C09046=1041.866,-97.475,-73.988,168.955,34.986,156.606
C09047=1041.872,-97.226,-73.998,168.958,34.986,156.606
C09048=1041.878,-96.977,-74.009,168.960,34.986,156.606
C09049=1041.883,-96.727,-74.019,168.962,34.986,156.606
C09050=1041.890,-96.477,-74.030,168.965,34.986,156.606
C09051=1041.895,-96.227,-74.040,168.967,34.986,156.606
C09052=1041.902,-95.978,-74.050,168.970,34.987,156.606
C09053=1041.908,-95.728,-74.061,168.972,34.987,156.606
C09054=1041.914,-95.478,-74.071,168.974,34.987,156.606
C09055=1041.920,-95.229,-74.082,168.977,34.987,156.606
C09056=1041.926,-94.979,-74.093,168.979,34.987,156.606
C09057=1041.932,-94.729,-74.102,168.982,34.987,156.606
C09058=1041.938,-94.479,-74.113,168.984,34.987,156.606
C09059=1041.945,-94.230,-74.124,168.986,34.987,156.606
C09060=1041.950,-93.980,-74.134,168.989,34.987,156.606
C09061=1041.956,-93.730,-74.145,168.991,34.987,156.606
C09062=1041.962,-93.481,-74.155,168.994,34.988,156.606
C09063=1041.969,-93.230,-74.165,168.996,34.988,156.606
C09064=1041.975,-92.981,-74.176,168.998,34.988,156.606
C09065=1041.981,-92.732,-74.187,169.001,34.988,156.606
C09066=1041.986,-92.482,-74.197,169.003,34.988,156.606
C09067=1041.993,-92.232,-74.207,169.006,34.988,156.606
C09068=1041.999,-91.982,-74.218,169.008,34.988,156.606
C09069=1042.005,-91.733,-74.229,169.011,34.988,156.606
C09070=1042.011,-91.484,-74.239,169.013,34.988,156.606
C09071=1042.017,-91.233,-74.250,169.015,34.988,156.606
C09072=1042.024,-90.984,-74.260,169.018,34.989,156.606
C09073=1042.029,-90.734,-74.271,169.020,34.989,156.606
C09074=1042.036,-90.485,-74.281,169.023,34.989,156.606
C09075=1042.042,-90.235,-74.293,169.025,34.989,156.606
C09076=1042.048,-89.985,-74.303,169.027,34.990,156.606
C09077=1042.054,-89.735,-74.313,169.030,34.990,156.606
C09078=1042.061,-89.485,-74.324,169.032,34.990,156.606
C09079=1042.066,-89.236,-74.335,169.034,34.990,156.606
C09080=1042.073,-88.987,-74.346,169.037,34.990,156.606
C09081=1042.079,-88.736,-74.357,169.039,34.990,156.606
C09082=1042.085,-88.487,-74.366,169.042,34.990,156.606
C09083=1042.091,-88.237,-74.377,169.044,34.990,156.606
C09084=1042.097,-87.987,-74.388,169.046,34.990,156.606
C09085=1042.104,-87.738,-74.399,169.049,34.991,156.606
C09086=1042.110,-87.488,-74.410,169.051,34.991,156.606
C09087=1042.116,-87.238,-74.421,169.054,34.991,156.606
C09088=1042.122,-86.989,-74.431,169.056,34.991,156.606
C09089=1042.128,-86.739,-74.442,169.058,34.991,156.606
C09090=1042.134,-86.489,-74.453,169.061,34.992,156.606
C09091=1042.141,-86.240,-74.464,169.063,34.992,156.606
C09092=1042.147,-85.991,-74.474,169.066,34.992,156.606
C09093=1042.153,-85.740,-74.486,169.068,34.992,156.606
C09094=1042.159,-85.491,-74.496,169.070,34.993,156.606
C09095=1042.166,-85.240,-74.506,169.073,34.993,156.606
C09096=1042.171,-84.991,-74.517,169.075,34.993,156.606
C09097=1042.178,-84.742,-74.528,169.077,34.993,156.606
C09098=1042.184,-84.492,-74.539,169.079,34.993,156.605
C09099=1042.190,-84.242,-74.550,169.081,34.993,156.605
C09100=1042.197,-83.957,-74.563,169.085,34.994,156.606
C09101=1042.204,-83.673,-74.575,169.087,34.994,156.606
C09102=1042.211,-83.387,-74.587,169.089,34.994,156.606
C09103=1042.219,-83.103,-74.600,169.092,34.994,156.605
C09104=1042.225,-82.853,-74.611,169.094,34.994,156.605
C09105=1042.231,-82.604,-74.621,169.097,34.995,156.606
C09106=1042.238,-82.354,-74.632,169.099,34.995,156.606
C09107=1042.243,-82.104,-74.643,169.102,34.995,156.605
C09108=1042.250,-81.854,-74.654,169.104,34.995,156.605
C09109=1042.256,-81.605,-74.665,169.106,34.995,156.605
C09110=1042.263,-81.355,-74.676,169.109,34.995,156.605
C09111=1042.269,-81.106,-74.686,169.111,34.996,156.606
C09112=1042.276,-80.856,-74.698,169.113,34.996,156.606
C09113=1042.281,-80.606,-74.709,169.116,34.996,156.605
C09114=1042.288,-80.356,-74.720,169.118,34.996,156.605
C09115=1042.294,-80.107,-74.731,169.121,34.997,156.606
C09116=1042.301,-79.857,-74.742,169.123,34.997,156.606
C09117=1042.306,-79.607,-74.753,169.125,34.997,156.606
C09118=1042.313,-79.357,-74.764,169.128,34.997,156.605
C09119=1042.319,-79.108,-74.776,169.130,34.998,156.606
C09120=1042.325,-78.858,-74.787,169.132,34.998,156.606
C09121=1042.331,-78.609,-74.798,169.135,34.999,156.606
C09122=1042.337,-78.358,-74.809,169.137,34.999,156.606
C09123=1042.343,-78.110,-74.821,169.139,34.999,156.606
C09124=1042.350,-77.859,-74.832,169.142,35.000,156.606
C09125=1042.356,-77.610,-74.842,169.144,35.000,156.606
C09126=1042.362,-77.360,-74.853,169.146,35.000,156.606
C09127=1042.368,-77.111,-74.865,169.149,35.001,156.606
C09128=1042.375,-76.861,-74.876,169.151,35.001,156.606
C09129=1042.381,-76.611,-74.887,169.153,35.002,156.606
C09130=1042.387,-76.362,-74.899,169.156,35.002,156.606
C09131=1042.393,-76.112,-74.910,169.158,35.002,156.606
C09132=1042.399,-75.862,-74.921,169.160,35.003,156.606
C09133=1042.406,-75.613,-74.933,169.163,35.003,156.606
C09134=1042.412,-75.363,-74.944,169.165,35.003,156.606
C09135=1042.418,-75.113,-74.955,169.167,35.004,156.606
C09136=1042.424,-74.864,-74.967,169.170,35.004,156.606
C09137=1042.430,-74.614,-74.978,169.172,35.004,156.606
C09138=1042.437,-74.364,-74.989,169.174,35.004,156.606
C09139=1042.443,-74.115,-75.001,169.176,35.005,156.606
C09140=1042.449,-73.865,-75.012,169.179,35.005,156.606
C09141=1042.455,-73.616,-75.024,169.181,35.006,156.606
C09142=1042.461,-73.365,-75.036,169.183,35.007,156.606
C09143=1042.466,-73.116,-75.047,169.186,35.007,156.606
C09144=1042.473,-72.866,-75.058,169.188,35.008,156.606
C09145=1042.479,-72.616,-75.070,169.190,35.008,156.606
C09146=1042.485,-72.367,-75.081,169.192,35.008,156.606
C09147=1042.491,-72.117,-75.093,169.195,35.009,156.606
C09148=1042.497,-71.868,-75.105,169.197,35.009,156.606
C09149=1042.503,-71.618,-75.116,169.199,35.010,156.606
C09150=1042.509,-71.369,-75.128,169.203,35.011,156.607
C09151=1042.515,-71.118,-75.139,169.204,35.011,156.607
C09152=1042.522,-70.869,-75.151,169.207,35.012,156.607
C09153=1042.528,-70.620,-75.163,169.209,35.012,156.607
C09154=1042.534,-70.370,-75.174,169.212,35.012,156.607
C09155=1042.539,-70.120,-75.186,169.214,35.013,156.607
C09156=1042.546,-69.870,-75.198,169.216,35.013,156.607
C09157=1042.552,-69.621,-75.210,169.219,35.014,156.607
C09158=1042.558,-69.371,-75.220,169.221,35.015,156.607
C09159=1042.564,-69.121,-75.233,169.223,35.015,156.607
C09160=1042.571,-68.872,-75.245,169.225,35.015,156.607
C09161=1042.576,-68.622,-75.256,169.228,35.016,156.607
C09162=1042.583,-68.373,-75.268,169.230,35.016,156.607
C09163=1042.589,-68.122,-75.280,169.232,35.017,156.607
C09164=1042.596,-67.840,-75.293,169.235,35.018,156.607
C09165=1042.602,-67.557,-75.306,169.237,35.018,156.607
C09166=1042.609,-67.275,-75.319,169.240,35.019,156.607
C09167=1042.616,-66.993,-75.333,169.242,35.019,156.607
C09168=1042.623,-66.742,-75.344,169.245,35.020,156.608
C09169=1042.629,-66.493,-75.356,169.247,35.020,156.608
C09170=1042.636,-66.243,-75.368,169.249,35.021,156.608
C09171=1042.641,-65.994,-75.380,169.251,35.022,156.608
C09172=1042.648,-65.744,-75.392,169.254,35.022,156.608
C09173=1042.654,-65.494,-75.404,169.256,35.022,156.608
C09174=1042.659,-65.245,-75.415,169.258,35.023,156.608
C09175=1042.666,-64.995,-75.427,169.260,35.023,156.608
C09176=1042.672,-64.745,-75.439,169.263,35.024,156.608
C09177=1042.679,-64.496,-75.451,169.265,35.025,156.608
C09178=1042.684,-64.246,-75.462,169.267,35.025,156.608
C09179=1042.691,-63.996,-75.474,169.270,35.026,156.608
C09180=1042.697,-63.747,-75.486,169.272,35.026,156.608
C09181=1042.703,-63.497,-75.499,169.274,35.027,156.608
C09182=1042.709,-63.248,-75.511,169.276,35.027,156.608
C09183=1042.716,-62.998,-75.522,169.279,35.028,156.608
C09184=1042.722,-62.748,-75.534,169.281,35.029,156.608
C09185=1042.728,-62.499,-75.546,169.283,35.029,156.609
C09186=1042.735,-62.249,-75.558,169.285,35.029,156.608
C09187=1042.740,-62.000,-75.570,169.288,35.030,156.609
C09188=1042.747,-61.750,-75.582,169.290,35.031,156.609
C09189=1042.753,-61.500,-75.594,169.292,35.031,156.609
C09190=1042.760,-61.250,-75.606,169.294,35.032,156.609
C09191=1042.766,-61.001,-75.618,169.296,35.032,156.609
C09192=1042.772,-60.752,-75.630,169.299,35.033,156.609
C09193=1042.778,-60.502,-75.642,169.301,35.033,156.609
C09194=1042.784,-60.252,-75.654,169.303,35.034,156.609
C09195=1042.791,-60.003,-75.666,169.305,35.035,156.609
C09196=1042.797,-59.752,-75.677,169.308,35.035,156.609
C09197=1042.803,-59.503,-75.690,169.310,35.035,156.609
C09198=1042.809,-59.254,-75.702,169.312,35.036,156.609
C09199=1042.816,-59.004,-75.714,169.314,35.037,156.609
C09200=1042.822,-58.754,-75.726,169.317,35.038,156.609
C09201=1042.829,-58.505,-75.738,169.319,35.038,156.609
C09202=1042.834,-58.255,-75.751,169.321,35.038,156.610
C09203=1042.841,-58.005,-75.763,169.323,35.039,156.610
C09204=1042.848,-57.756,-75.775,169.326,35.040,156.610
C09205=1042.854,-57.506,-75.787,169.328,35.041,156.610
C09206=1042.860,-57.257,-75.799,169.330,35.041,156.610
C09207=1042.866,-57.007,-75.811,169.332,35.041,156.610
C09208=1042.872,-56.757,-75.823,169.334,35.042,156.610
C09209=1042.879,-56.508,-75.835,169.337,35.043,156.610
C09210=1042.886,-56.258,-75.847,169.339,35.043,156.610
C09211=1042.891,-56.008,-75.860,169.341,35.044,156.610
C09212=1042.898,-55.759,-75.872,169.343,35.044,156.610
C09213=1042.904,-55.509,-75.884,169.346,35.045,156.610
C09214=1042.911,-55.259,-75.896,169.348,35.046,156.610
C09215=1042.917,-55.010,-75.908,169.350,35.046,156.610
C09216=1042.923,-54.760,-75.921,169.352,35.047,156.610
C09217=1042.930,-54.510,-75.933,169.354,35.047,156.611
C09218=1042.936,-54.261,-75.945,169.358,35.048,156.611
C09219=1042.942,-54.011,-75.957,169.360,35.049,156.611
C09220=1042.949,-53.762,-75.970,169.362,35.049,156.611
C09221=1042.955,-53.512,-75.982,169.364,35.050,156.611
C09222=1042.962,-53.262,-75.994,169.367,35.050,156.611
C09223=1042.969,-53.013,-76.006,169.369,35.051,156.611
C09224=1042.974,-52.763,-76.019,169.371,35.052,156.611
C09225=1042.981,-52.513,-76.031,169.373,35.052,156.611
C09226=1042.987,-52.264,-76.043,169.375,35.053,156.611
C09227=1042.994,-52.014,-76.055,169.378,35.053,156.611
C09228=1043.000,-51.733,-76.069,169.380,35.054,156.611
C09229=1043.008,-51.452,-76.084,169.383,35.055,156.611
C09230=1043.016,-51.170,-76.097,169.385,35.056,156.612
C09231=1043.023,-50.889,-76.111,169.388,35.056,156.612
C09232=1043.030,-50.639,-76.123,169.390,35.057,156.612
C09233=1043.035,-50.389,-76.136,169.392,35.057,156.612
C09234=1043.042,-50.140,-76.149,169.394,35.058,156.612
C09235=1043.048,-49.890,-76.162,169.396,35.059,156.612
C09236=1043.054,-49.641,-76.174,169.398,35.060,156.612
C09237=1043.060,-49.391,-76.186,169.401,35.061,156.612
C09238=1043.066,-49.141,-76.199,169.403,35.061,156.612
C09239=1043.073,-48.892,-76.211,169.405,35.062,156.612
C09240=1043.079,-48.642,-76.224,169.407,35.063,156.612
C09241=1043.085,-48.393,-76.237,169.409,35.064,156.613
C09242=1043.091,-48.143,-76.250,169.411,35.064,156.613
C09243=1043.098,-47.893,-76.262,169.413,35.065,156.613
C09244=1043.104,-47.644,-76.275,169.416,35.066,156.613
C09245=1043.110,-47.394,-76.288,169.418,35.066,156.613
C09246=1043.116,-47.144,-76.300,169.420,35.067,156.613
C09247=1043.123,-46.895,-76.313,169.422,35.068,156.613
C09248=1043.129,-46.645,-76.325,169.424,35.069,156.613
C09249=1043.135,-46.396,-76.339,169.426,35.070,156.613
C09250=1043.141,-46.146,-76.351,169.429,35.071,156.614
C09251=1043.147,-45.896,-76.364,169.431,35.071,156.614
C09252=1043.154,-45.647,-76.376,169.433,35.072,156.614
C09253=1043.159,-45.397,-76.389,169.435,35.073,156.614
C09254=1043.166,-45.148,-76.402,169.437,35.074,156.614
C09255=1043.172,-44.898,-76.415,169.440,35.074,156.614
C09256=1043.179,-44.649,-76.427,169.442,35.075,156.614
C09257=1043.184,-44.400,-76.440,169.445,35.076,156.614
C09258=1043.191,-44.150,-76.453,169.447,35.076,156.614
C09259=1043.197,-43.900,-76.466,169.449,35.077,156.614
C09260=1043.203,-43.650,-76.479,169.451,35.078,156.615
C09261=1043.210,-43.401,-76.491,169.453,35.079,156.615
C09262=1043.216,-43.152,-76.505,169.455,35.080,156.615
C09263=1043.222,-42.902,-76.517,169.457,35.081,156.615
C09264=1043.228,-42.652,-76.531,169.459,35.081,156.615
C09265=1043.235,-42.403,-76.542,169.462,35.082,156.615
C09266=1043.241,-42.154,-76.556,169.464,35.083,156.615
C09267=1043.248,-41.903,-76.569,169.466,35.084,156.615
C09268=1043.254,-41.654,-76.582,169.468,35.084,156.615
C09269=1043.260,-41.404,-76.595,169.470,35.086,156.616
C09270=1043.267,-41.155,-76.607,169.472,35.086,156.616
C09271=1043.273,-40.905,-76.620,169.474,35.087,156.616
C09272=1043.279,-40.656,-76.633,169.476,35.088,156.616
C09273=1043.286,-40.406,-76.647,169.479,35.088,156.616
C09274=1043.292,-40.156,-76.659,169.481,35.089,156.616
C09275=1043.298,-39.907,-76.672,169.483,35.090,156.616
C09276=1043.305,-39.657,-76.684,169.485,35.091,156.616
C09277=1043.311,-39.408,-76.698,169.487,35.091,156.616
C09278=1043.318,-39.158,-76.711,169.489,35.093,156.616
C09279=1043.323,-38.908,-76.724,169.491,35.093,156.617
C09280=1043.330,-38.659,-76.737,169.493,35.094,156.617
C09281=1043.336,-38.409,-76.750,169.495,35.095,156.617
C09282=1043.342,-38.160,-76.763,169.498,35.096,156.617
C09283=1043.349,-37.910,-76.777,169.500,35.097,156.617
C09284=1043.355,-37.660,-76.790,169.503,35.098,156.617
C09285=1043.361,-37.410,-76.802,169.505,35.098,156.617
C09286=1043.367,-37.161,-76.816,169.507,35.100,156.617
C09287=1043.373,-36.912,-76.829,169.509,35.100,156.618
C09288=1043.380,-36.662,-76.843,169.511,35.101,156.618
C09289=1043.386,-36.412,-76.855,169.513,35.102,156.618
C09290=1043.392,-36.163,-76.868,169.515,35.103,156.618
C09291=1043.398,-35.914,-76.882,169.517,35.104,156.618
C09292=1043.405,-35.632,-76.897,169.520,35.105,156.618
C09293=1043.412,-35.352,-76.912,169.522,35.106,156.618
C09294=1043.420,-35.071,-76.927,169.524,35.107,156.618
C09295=1043.426,-34.789,-76.942,169.527,35.108,156.619
C09296=1043.433,-34.540,-76.955,169.529,35.109,156.619
C09297=1043.439,-34.291,-76.968,169.531,35.110,156.619
C09298=1043.445,-34.041,-76.981,169.533,35.111,156.619
C09299=1043.452,-33.791,-76.995,169.535,35.112,156.619
C09300=1043.458,-33.542,-77.008,169.537,35.112,156.619
C09301=1043.464,-33.292,-77.021,169.539,35.114,156.619
C09302=1043.470,-33.043,-77.034,169.541,35.114,156.620
C09303=1043.477,-32.793,-77.048,169.543,35.115,156.620
C09304=1043.483,-32.544,-77.061,169.545,35.116,156.620
C09305=1043.489,-32.294,-77.075,169.547,35.117,156.620
C09306=1043.495,-32.044,-77.089,169.549,35.118,156.620
C09307=1043.502,-31.795,-77.102,169.552,35.119,156.620
C09308=1043.508,-31.546,-77.115,169.554,35.120,156.620
C09309=1043.514,-31.295,-77.128,169.557,35.121,156.620
C09310=1043.521,-31.046,-77.141,169.559,35.122,156.621
C09311=1043.527,-30.797,-77.155,169.561,35.123,156.621
C09312=1043.534,-30.547,-77.168,169.563,35.123,156.621
C09313=1043.540,-30.297,-77.182,169.565,35.125,156.621
C09314=1043.546,-30.048,-77.195,169.567,35.125,156.621
C09315=1043.552,-29.798,-77.209,169.569,35.126,156.621
C09316=1043.558,-29.549,-77.222,169.571,35.127,156.621
C09317=1043.565,-29.299,-77.236,169.573,35.128,156.622
C09318=1043.571,-29.049,-77.249,169.575,35.129,156.622
C09319=1043.578,-28.800,-77.262,169.577,35.130,156.622
C09320=1043.584,-28.551,-77.276,169.579,35.131,156.622
C09321=1043.591,-28.301,-77.289,169.581,35.132,156.622
C09322=1043.597,-28.052,-77.303,169.583,35.132,156.622
C09323=1043.603,-27.801,-77.317,169.585,35.134,156.622
C09324=1043.609,-27.552,-77.330,169.587,35.134,156.622
C09325=1043.615,-27.303,-77.343,169.589,35.135,156.623
C09326=1043.622,-27.053,-77.357,169.591,35.136,156.623
C09327=1043.629,-26.804,-77.371,169.593,35.137,156.623
C09328=1043.634,-26.555,-77.385,169.595,35.139,156.623
C09329=1043.641,-26.305,-77.399,169.598,35.139,156.623
C09330=1043.647,-26.055,-77.412,169.600,35.141,156.623
C09331=1043.653,-25.805,-77.426,169.602,35.141,156.623
C09332=1043.659,-25.556,-77.439,169.604,35.143,156.624
C09333=1043.666,-25.307,-77.453,169.606,35.143,156.624
C09334=1043.672,-25.056,-77.467,169.608,35.145,156.624
C09335=1043.678,-24.808,-77.481,169.611,35.145,156.624
C09336=1043.685,-24.558,-77.494,169.613,35.147,156.624
C09337=1043.691,-24.308,-77.508,169.615,35.147,156.624
C09338=1043.697,-24.059,-77.522,169.617,35.149,156.625
C09339=1043.703,-23.809,-77.536,169.619,35.150,156.625
C09340=1043.709,-23.560,-77.550,169.621,35.151,156.625
C09341=1043.716,-23.310,-77.563,169.623,35.152,156.625
C09342=1043.722,-23.060,-77.577,169.625,35.153,156.625
C09343=1043.728,-22.811,-77.591,169.627,35.154,156.625
C09344=1043.735,-22.562,-77.605,169.629,35.155,156.626
C09345=1043.740,-22.312,-77.619,169.631,35.156,156.626
C09346=1043.747,-22.062,-77.632,169.633,35.157,156.626
C09347=1043.753,-21.813,-77.646,169.635,35.158,156.626
C09348=1043.760,-21.563,-77.661,169.637,35.159,156.626
C09349=1043.766,-21.314,-77.674,169.639,35.160,156.626
C09350=1043.772,-21.064,-77.688,169.641,35.161,156.626
C09351=1043.778,-20.815,-77.701,169.643,35.162,156.627
C09352=1043.785,-20.565,-77.716,169.645,35.163,156.627
C09353=1043.791,-20.316,-77.730,169.647,35.164,156.627
C09354=1043.798,-20.066,-77.743,169.649,35.165,156.627
C09355=1043.804,-19.817,-77.758,169.651,35.166,156.627
C09356=1043.811,-19.534,-77.773,169.654,35.167,156.627
C09357=1043.818,-19.253,-77.789,169.656,35.169,156.628
C09358=1043.825,-18.971,-77.805,169.658,35.169,156.628
C09359=1043.832,-18.690,-77.821,169.660,35.171,156.628
C09360=1043.839,-18.440,-77.834,169.662,35.172,156.628
C09361=1043.844,-18.191,-77.848,169.664,35.173,156.628
C09362=1043.852,-17.941,-77.863,169.666,35.174,156.628
C09363=1043.858,-17.691,-77.877,169.668,35.175,156.629
C09364=1043.864,-17.442,-77.890,169.670,35.176,156.629
C09365=1043.871,-17.192,-77.904,169.672,35.177,156.629
C09366=1043.876,-16.943,-77.918,169.675,35.178,156.629
C09367=1043.884,-16.693,-77.933,169.677,35.179,156.629
C09368=1043.889,-16.444,-77.947,169.679,35.180,156.629
C09369=1043.896,-16.195,-77.961,169.681,35.181,156.629
C09370=1043.902,-15.945,-77.975,169.683,35.182,156.630
C09371=1043.908,-15.695,-77.988,169.685,35.183,156.630
C09372=1043.916,-15.446,-78.003,169.687,35.184,156.630
C09373=1043.921,-15.196,-78.017,169.689,35.185,156.630
C09374=1043.927,-14.946,-78.032,169.691,35.186,156.630
C09375=1043.934,-14.697,-78.045,169.693,35.188,156.631
C09376=1043.940,-14.448,-78.060,169.695,35.188,156.631
C09377=1043.946,-14.199,-78.074,169.697,35.190,156.631
C09378=1043.953,-13.949,-78.088,169.699,35.191,156.631
C09379=1043.959,-13.699,-78.103,169.701,35.192,156.631
C09380=1043.965,-13.449,-78.117,169.703,35.193,156.631
C09381=1043.972,-13.200,-78.131,169.705,35.194,156.632
C09382=1043.977,-12.950,-78.145,169.706,35.195,156.632
C09383=1043.983,-12.701,-78.160,169.709,35.196,156.632
C09384=1043.990,-12.452,-78.174,169.711,35.198,156.632
C09385=1043.996,-12.202,-78.188,169.713,35.198,156.632
C09386=1044.002,-11.952,-78.203,169.715,35.200,156.632
C09387=1044.009,-11.703,-78.216,169.717,35.201,156.633
C09388=1044.015,-11.453,-78.231,169.719,35.202,156.633
C09389=1044.021,-11.204,-78.246,169.721,35.203,156.633
C09390=1044.028,-10.954,-78.260,169.723,35.204,156.633
C09391=1044.034,-10.705,-78.275,169.725,35.205,156.633
C09392=1044.040,-10.456,-78.289,169.727,35.206,156.633
C09393=1044.047,-10.206,-78.303,169.729,35.208,156.634
C09394=1044.053,-9.956,-78.318,169.731,35.209,156.634
C09395=1044.059,-9.707,-78.332,169.733,35.210,156.634
C09396=1044.066,-9.457,-78.346,169.734,35.211,156.634
C09397=1044.072,-9.208,-78.361,169.736,35.212,156.634
C09398=1044.078,-8.959,-78.375,169.739,35.213,156.634
C09399=1044.084,-8.709,-78.390,169.741,35.215,156.635
C09400=1044.091,-8.459,-78.404,169.743,35.215,156.635
C09401=1044.097,-8.210,-78.419,169.745,35.217,156.635
C09402=1044.103,-7.960,-78.434,169.747,35.218,156.635
C09403=1044.110,-7.710,-78.447,169.749,35.219,156.635
C09404=1044.116,-7.461,-78.462,169.751,35.220,156.636
C09405=1044.122,-7.212,-78.477,169.753,35.221,156.636
C09406=1044.129,-6.962,-78.492,169.755,35.223,156.636
C09407=1044.135,-6.714,-78.506,169.757,35.223,156.636
C09408=1044.141,-6.463,-78.520,169.759,35.225,156.636
C09409=1044.147,-6.214,-78.535,169.760,35.226,156.636
C09410=1044.155,-5.964,-78.549,169.762,35.227,156.637
C09411=1044.160,-5.715,-78.564,169.764,35.228,156.637
C09412=1044.167,-5.466,-78.579,169.766,35.229,156.637
C09413=1044.173,-5.215,-78.593,169.768,35.230,156.637
C09414=1044.180,-4.966,-78.607,169.771,35.231,156.637
C09415=1044.186,-4.717,-78.622,169.773,35.233,156.638
C09416=1044.192,-4.467,-78.637,169.775,35.233,156.638
C09417=1044.199,-4.218,-78.652,169.777,35.235,156.638
C09418=1044.206,-3.968,-78.666,169.779,35.236,156.638
C09419=1044.211,-3.719,-78.681,169.780,35.237,156.638
C09420=1044.219,-3.436,-78.697,169.783,35.238,156.638
C09421=1044.226,-3.152,-78.713,169.785,35.239,156.639
C09422=1044.232,-2.869,-78.731,169.787,35.241,156.639
C09423=1044.239,-2.586,-78.747,169.789,35.243,156.639
C09424=1044.246,-2.336,-78.762,169.791,35.244,156.639
C09425=1044.252,-2.087,-78.777,169.793,35.245,156.639
C09426=1044.258,-1.837,-78.792,169.795,35.246,156.640
C09427=1044.264,-1.588,-78.807,169.797,35.247,156.640
C09428=1044.271,-1.338,-78.822,169.799,35.249,156.640
C09429=1044.277,-1.089,-78.837,169.801,35.250,156.640
C09430=1044.283,-0.839,-78.852,169.803,35.251,156.641
C09431=1044.289,-0.590,-78.866,169.805,35.253,156.641
C09432=1044.296,-0.340,-78.881,169.807,35.254,156.641
C09433=1044.302,-0.091,-78.896,169.809,35.255,156.641
C09434=1044.308,0.159,-78.911,169.810,35.256,156.641
C09435=1044.314,0.408,-78.926,169.812,35.257,156.641
C09436=1044.320,0.658,-78.941,169.814,35.259,156.642
C09437=1044.326,0.908,-78.956,169.816,35.260,156.642
C09438=1044.333,1.157,-78.972,169.818,35.261,156.642
C09439=1044.339,1.406,-78.986,169.820,35.263,156.642
C09440=1044.345,1.655,-79.001,169.822,35.263,156.642
C09441=1044.351,1.905,-79.016,169.824,35.265,156.643
C09442=1044.358,2.155,-79.031,169.826,35.266,156.643
C09443=1044.364,2.404,-79.046,169.828,35.267,156.643
C09444=1044.371,2.654,-79.061,169.830,35.269,156.643
C09445=1044.376,2.903,-79.076,169.832,35.270,156.644
C09446=1044.383,3.152,-79.091,169.834,35.271,156.644
C09447=1044.389,3.402,-79.106,169.835,35.273,156.644
C09448=1044.396,3.651,-79.121,169.837,35.273,156.644
C09449=1044.402,3.901,-79.136,169.839,35.275,156.644
C09450=1044.408,4.151,-79.152,169.841,35.276,156.644
C09451=1044.414,4.400,-79.166,169.843,35.277,156.645
C09452=1044.420,4.649,-79.181,169.845,35.279,156.645
C09453=1044.427,4.898,-79.197,169.847,35.280,156.645
C09454=1044.433,5.148,-79.212,169.849,35.281,156.645
C09455=1044.439,5.398,-79.227,169.851,35.283,156.646
C09456=1044.446,5.647,-79.242,169.853,35.283,156.646
C09457=1044.452,5.897,-79.257,169.855,35.285,156.646
C09458=1044.458,6.145,-79.272,169.857,35.286,156.646
C09459=1044.465,6.395,-79.287,169.859,35.287,156.646
C09460=1044.471,6.645,-79.302,169.860,35.288,156.647
C09461=1044.477,6.895,-79.317,169.862,35.290,156.647
C09462=1044.483,7.144,-79.333,169.864,35.291,156.647
C09463=1044.490,7.393,-79.348,169.866,35.292,156.647
C09464=1044.496,7.643,-79.363,169.868,35.293,156.647
C09465=1044.503,7.892,-79.379,169.870,35.294,156.648
C09466=1044.509,8.142,-79.394,169.871,35.296,156.648
C09467=1044.516,8.391,-79.409,169.874,35.297,156.648
C09468=1044.522,8.641,-79.423,169.876,35.298,156.648
C09469=1044.529,8.890,-79.439,169.878,35.300,156.648
C09470=1044.534,9.139,-79.454,169.880,35.301,156.649
C09471=1044.540,9.389,-79.469,169.882,35.302,156.649
C09472=1044.547,9.638,-79.485,169.883,35.303,156.649
C09473=1044.553,9.888,-79.500,169.885,35.304,156.649
C09474=1044.560,10.137,-79.515,169.887,35.306,156.649
C09475=1044.566,10.386,-79.530,169.889,35.307,156.650
C09476=1044.573,10.636,-79.545,169.891,35.308,156.650
C09477=1044.579,10.885,-79.561,169.893,35.310,156.650
C09478=1044.585,11.135,-79.577,169.894,35.310,156.650
C09479=1044.591,11.385,-79.592,169.896,35.312,156.650
C09480=1044.598,11.634,-79.607,169.899,35.313,156.651
C09481=1044.604,11.883,-79.622,169.901,35.314,156.651
C09482=1044.611,12.132,-79.638,169.903,35.316,156.651
C09483=1044.617,12.382,-79.653,169.904,35.317,156.651
C09484=1044.625,12.667,-79.670,169.907,35.318,156.651
C09485=1044.633,12.953,-79.688,169.909,35.320,156.652
C09486=1044.639,13.238,-79.706,169.911,35.321,156.652
C09487=1044.647,13.524,-79.723,169.913,35.322,156.652
C09488=1044.653,13.773,-79.739,169.915,35.324,156.652
C09489=1044.660,14.023,-79.754,169.916,35.325,156.652
C09490=1044.666,14.272,-79.770,169.918,35.326,156.653
C09491=1044.672,14.522,-79.785,169.920,35.328,156.653
C09492=1044.679,14.771,-79.801,169.923,35.329,156.653
C09493=1044.685,15.020,-79.816,169.925,35.330,156.653
C09494=1044.691,15.270,-79.832,169.926,35.331,156.654
C09495=1044.698,15.519,-79.848,169.928,35.333,156.654
C09496=1044.703,15.769,-79.863,169.930,35.334,156.654
C09497=1044.710,16.018,-79.879,169.932,35.335,156.654
C09498=1044.716,16.267,-79.894,169.934,35.337,156.654
C09499=1044.722,16.517,-79.910,169.935,35.338,156.655
C09500=1044.729,16.766,-79.925,169.937,35.339,156.655
C09501=1044.735,17.016,-79.941,169.939,35.341,156.655
C09502=1044.741,17.265,-79.957,169.941,35.342,156.655
C09503=1044.748,17.514,-79.972,169.943,35.343,156.656
C09504=1044.754,17.764,-79.988,169.945,35.345,156.656
C09505=1044.760,18.013,-80.004,169.947,35.346,156.656
C09506=1044.766,18.263,-80.019,169.949,35.347,156.656
C09507=1044.773,18.512,-80.035,169.951,35.349,156.656
C09508=1044.779,18.761,-80.051,169.952,35.350,156.657
C09509=1044.785,19.011,-80.066,169.954,35.351,156.657
C09510=1044.792,19.260,-80.082,169.956,35.353,156.657
C09511=1044.798,19.510,-80.099,169.958,35.354,156.657
C09512=1044.804,19.750,-80.113,169.959,35.355,156.657
C09513=1044.810,19.991,-80.128,169.961,35.356,156.658
C09514=1044.817,20.231,-80.143,169.963,35.358,156.658
C09515=1044.822,20.472,-80.159,169.966,35.359,156.658
C09516=1044.829,20.712,-80.174,169.967,35.360,156.658
C09517=1044.834,20.953,-80.189,169.969,35.362,156.659
C09518=1044.840,21.193,-80.204,169.971,35.363,156.659
C09519=1044.847,21.434,-80.220,169.972,35.364,156.659
C09520=1044.853,21.683,-80.235,169.974,35.366,156.659
C09521=1044.859,21.933,-80.252,169.976,35.367,156.659
C09522=1044.865,22.182,-80.268,169.978,35.368,156.660
C09523=1044.872,22.432,-80.283,169.979,35.370,156.660
C09524=1044.877,22.681,-80.299,169.981,35.371,156.660
C09525=1044.885,22.931,-80.315,169.983,35.372,156.660
C09526=1044.891,23.180,-80.331,169.986,35.374,156.661
C09527=1044.897,23.429,-80.347,169.987,35.375,156.661
C09528=1044.903,23.679,-80.363,169.989,35.376,156.661
C09529=1044.910,23.928,-80.378,169.991,35.377,156.661
C09530=1044.916,24.177,-80.394,169.993,35.379,156.661
C09531=1044.922,24.427,-80.411,169.994,35.380,156.662
C09532=1044.929,24.677,-80.427,169.996,35.381,156.662
C09533=1044.935,24.926,-80.443,169.998,35.383,156.662
C09534=1044.942,25.175,-80.459,170.000,35.384,156.662
C09535=1044.947,25.425,-80.474,170.001,35.385,156.663
C09536=1044.954,25.674,-80.490,170.003,35.387,156.663
C09537=1044.960,25.923,-80.506,170.006,35.388,156.663
C09538=1044.966,26.173,-80.523,170.008,35.390,156.663
C09539=1044.973,26.422,-80.538,170.009,35.391,156.664
C09540=1044.979,26.672,-80.555,170.011,35.392,156.664
C09541=1044.986,26.921,-80.570,170.013,35.394,156.664
C09542=1044.992,27.170,-80.587,170.015,35.395,156.664
C09543=1044.998,27.419,-80.603,170.016,35.396,156.664
C09544=1045.005,27.669,-80.619,170.018,35.398,156.665
C09545=1045.011,27.919,-80.635,170.020,35.399,156.665
C09546=1045.017,28.168,-80.651,170.022,35.400,156.665
C09547=1045.024,28.417,-80.667,170.023,35.402,156.665
C09548=1045.031,28.722,-80.687,170.026,35.404,156.666
C09549=1045.038,29.026,-80.707,170.029,35.405,156.666
C09550=1045.046,29.330,-80.726,170.031,35.407,156.666
C09551=1045.054,29.635,-80.746,170.033,35.409,156.666
C09552=1045.060,29.884,-80.762,170.035,35.410,156.667
C09553=1045.066,30.133,-80.779,170.036,35.411,156.667
C09554=1045.072,30.383,-80.795,170.038,35.413,156.667
C09555=1045.079,30.632,-80.811,170.040,35.414,156.667
C09556=1045.085,30.882,-80.827,170.041,35.415,156.668
C09557=1045.091,31.131,-80.844,170.044,35.417,156.668
C09558=1045.097,31.380,-80.860,170.046,35.419,156.668
C09559=1045.104,31.630,-80.877,170.048,35.420,156.668
C09560=1045.111,31.879,-80.893,170.049,35.421,156.669
C09561=1045.117,32.128,-80.909,170.051,35.422,156.669
C09562=1045.123,32.378,-80.925,170.053,35.424,156.669
C09563=1045.129,32.628,-80.942,170.054,35.425,156.669
C09564=1045.135,32.877,-80.958,170.056,35.427,156.670
C09565=1045.142,33.126,-80.974,170.058,35.428,156.670
C09566=1045.148,33.375,-80.990,170.060,35.430,156.670
C09567=1045.155,33.625,-81.007,170.061,35.431,156.670
C09568=1045.160,33.874,-81.024,170.064,35.432,156.670
C09569=1045.166,34.123,-81.040,170.066,35.434,156.671
C09570=1045.173,34.374,-81.057,170.068,35.435,156.671
C09571=1045.180,34.623,-81.072,170.069,35.437,156.671
C09572=1045.186,34.871,-81.089,170.071,35.438,156.671
C09573=1045.192,35.121,-81.105,170.073,35.439,156.672
C09574=1045.198,35.371,-81.122,170.074,35.441,156.672
C09575=1045.204,35.620,-81.138,170.076,35.442,156.672
C09576=1045.210,35.869,-81.155,170.078,35.443,156.672
C09577=1045.218,36.119,-81.171,170.080,35.445,156.673
C09578=1045.224,36.368,-81.188,170.082,35.446,156.673
C09579=1045.230,36.617,-81.204,170.084,35.448,156.673
C09580=1045.236,36.867,-81.220,170.086,35.449,156.673
C09581=1045.243,37.116,-81.237,170.087,35.450,156.674
C09582=1045.249,37.365,-81.254,170.089,35.452,156.674
C09583=1045.255,37.615,-81.270,170.091,35.453,156.674
C09584=1045.261,37.864,-81.287,170.093,35.454,156.674
C09585=1045.267,38.113,-81.304,170.094,35.456,156.675
C09586=1045.274,38.364,-81.320,170.096,35.458,156.675
C09587=1045.280,38.612,-81.337,170.098,35.459,156.675
C09588=1045.286,38.862,-81.353,170.100,35.460,156.675
C09589=1045.293,39.112,-81.370,170.102,35.461,156.675
C09590=1045.299,39.360,-81.387,170.104,35.463,156.676
C09591=1045.305,39.610,-81.403,170.105,35.465,156.676
C09592=1045.312,39.859,-81.421,170.107,35.466,156.676
C09593=1045.318,40.109,-81.437,170.109,35.467,156.676
C09594=1045.324,40.358,-81.453,170.110,35.469,156.677
C09595=1045.330,40.607,-81.470,170.112,35.471,156.677
C09596=1045.336,40.857,-81.487,170.114,35.472,156.677
C09597=1045.343,41.105,-81.504,170.117,35.473,156.677
C09598=1045.349,41.355,-81.520,170.118,35.475,156.678
C09599=1045.355,41.605,-81.537,170.120,35.476,156.678
C09600=1045.361,41.853,-81.554,170.122,35.478,156.678
C09601=1045.367,42.104,-81.571,170.123,35.479,156.678
C09602=1045.374,42.353,-81.588,170.125,35.480,156.679
C09603=1045.380,42.603,-81.604,170.127,35.482,156.679
C09604=1045.386,42.851,-81.621,170.128,35.483,156.679
C09605=1045.392,43.101,-81.638,170.130,35.485,156.679
C09606=1045.399,43.350,-81.655,170.132,35.486,156.680
C09607=1045.405,43.599,-81.671,170.134,35.488,156.680
C09608=1045.412,43.849,-81.689,170.136,35.489,156.680
C09609=1045.417,44.099,-81.705,170.138,35.491,156.680
C09610=1045.423,44.347,-81.722,170.139,35.492,156.681
C09611=1045.430,44.597,-81.739,170.141,35.494,156.681
C09612=1045.437,44.883,-81.759,170.143,35.496,156.681
C09613=1045.444,45.170,-81.778,170.145,35.497,156.682
C09614=1045.451,45.456,-81.798,170.147,35.499,156.682
C09615=1045.458,45.743,-81.818,170.150,35.501,156.682
C09616=1045.464,45.992,-81.835,170.151,35.502,156.683
C09617=1045.471,46.242,-81.851,170.153,35.503,156.683
C09618=1045.476,46.491,-81.869,170.155,35.505,156.683
C09619=1045.482,46.740,-81.886,170.156,35.507,156.683
C09620=1045.489,46.990,-81.902,170.158,35.509,156.684
C09621=1045.494,47.239,-81.920,170.160,35.510,156.684
C09622=1045.501,47.488,-81.937,170.161,35.511,156.684
C09623=1045.507,47.737,-81.954,170.163,35.513,156.684
C09624=1045.513,47.986,-81.971,170.166,35.514,156.685
C09625=1045.520,48.236,-81.989,170.167,35.516,156.685
C09626=1045.526,48.485,-82.005,170.169,35.518,156.685
C09627=1045.532,48.735,-82.023,170.171,35.519,156.685
C09628=1045.538,48.984,-82.040,170.172,35.520,156.686
C09629=1045.545,49.234,-82.056,170.174,35.522,156.686
C09630=1045.550,49.483,-82.074,170.176,35.523,156.686
C09631=1045.557,49.732,-82.091,170.177,35.525,156.686
C09632=1045.563,49.982,-82.107,170.179,35.526,156.687
C09633=1045.569,50.231,-82.125,170.182,35.528,156.687
C09634=1045.575,50.480,-82.142,170.183,35.529,156.687
C09635=1045.581,50.729,-82.160,170.185,35.531,156.687
C09636=1045.587,50.979,-82.177,170.187,35.532,156.688
C09637=1045.594,51.228,-82.194,170.188,35.534,156.688
C09638=1045.600,51.478,-82.211,170.190,35.535,156.688
C09639=1045.606,51.726,-82.228,170.192,35.537,156.689
C09640=1045.613,51.976,-82.246,170.193,35.538,156.689
C09641=1045.618,52.225,-82.263,170.195,35.540,156.689
C09642=1045.625,52.475,-82.280,170.198,35.542,156.689
C09643=1045.632,52.724,-82.297,170.199,35.543,156.690
C09644=1045.637,52.973,-82.315,170.201,35.544,156.690
C09645=1045.644,53.223,-82.332,170.203,35.545,156.690
C09646=1045.650,53.472,-82.350,170.204,35.547,156.690
C09647=1045.656,53.722,-82.366,170.206,35.549,156.691
C09648=1045.662,53.971,-82.383,170.208,35.550,156.691
C09649=1045.669,54.220,-82.401,170.209,35.552,156.691
C09650=1045.675,54.469,-82.418,170.211,35.553,156.691
C09651=1045.682,54.719,-82.436,170.214,35.554,156.692
C09652=1045.687,54.968,-82.453,170.215,35.556,156.692
C09653=1045.694,55.217,-82.471,170.217,35.558,156.692
C09654=1045.700,55.467,-82.488,170.219,35.559,156.692
C09655=1045.706,55.716,-82.505,170.220,35.560,156.693
C09656=1045.713,55.966,-82.522,170.222,35.562,156.693
C09657=1045.719,56.215,-82.540,170.224,35.563,156.693
C09658=1045.725,56.464,-82.557,170.225,35.565,156.693
C09659=1045.731,56.714,-82.575,170.228,35.567,156.694
C09660=1045.738,56.962,-82.592,170.230,35.568,156.694
C09661=1045.745,57.212,-82.609,170.231,35.569,156.694
C09662=1045.750,57.461,-82.627,170.233,35.570,156.694
C09663=1045.757,57.710,-82.644,170.235,35.572,156.695
C09664=1045.763,57.960,-82.662,170.236,35.574,156.695
C09665=1045.769,58.209,-82.679,170.238,35.575,156.695
C09666=1045.776,58.458,-82.696,170.240,35.576,156.695
C09667=1045.782,58.707,-82.714,170.241,35.578,156.696
C09668=1045.789,58.957,-82.731,170.244,35.579,156.696
C09669=1045.795,59.206,-82.749,170.246,35.581,156.696
C09670=1045.801,59.455,-82.766,170.247,35.582,156.696
C09671=1045.808,59.705,-82.784,170.249,35.584,156.697
C09672=1045.814,59.954,-82.801,170.251,35.585,156.697
C09673=1045.820,60.203,-82.818,170.252,35.587,156.697
C09674=1045.826,60.453,-82.836,170.254,35.588,156.698
C09675=1045.833,60.702,-82.854,170.256,35.590,156.698
C09676=1045.840,60.988,-82.874,170.258,35.591,156.698
C09677=1045.848,61.275,-82.894,170.261,35.593,156.698
C09678=1045.855,61.561,-82.914,170.263,35.595,156.699
C09679=1045.862,61.847,-82.934,170.265,35.596,156.699
C09680=1045.868,62.096,-82.951,170.266,35.597,156.699
C09681=1045.875,62.345,-82.970,170.268,35.599,156.699
C09682=1045.882,62.595,-82.987,170.270,35.601,156.700
C09683=1045.888,62.843,-83.004,170.271,35.602,156.700
C09684=1045.894,63.093,-83.022,170.273,35.603,156.700
C09685=1045.901,63.343,-83.039,170.276,35.605,156.701
C09686=1045.907,63.592,-83.057,170.277,35.606,156.701
C09687=1045.913,63.841,-83.074,170.279,35.608,156.701
C09688=1045.920,64.091,-83.092,170.281,35.609,156.701
C09689=1045.926,64.340,-83.111,170.282,35.611,156.702
C09690=1045.932,64.589,-83.128,170.284,35.612,156.702
C09691=1045.938,64.838,-83.146,170.286,35.614,156.702
C09692=1045.944,65.088,-83.164,170.287,35.615,156.702
C09693=1045.951,65.337,-83.181,170.289,35.617,156.703
C09694=1045.957,65.586,-83.199,170.291,35.619,156.703
C09695=1045.963,65.836,-83.217,170.293,35.620,156.703
C09696=1045.970,66.085,-83.235,170.295,35.621,156.703
C09697=1045.976,66.334,-83.253,170.296,35.623,156.704
C09698=1045.982,66.583,-83.271,170.298,35.624,156.704
C09699=1045.989,66.833,-83.288,170.300,35.626,156.704
C09700=1045.994,67.082,-83.306,170.301,35.628,156.704
C09701=1046.001,67.331,-83.324,170.303,35.629,156.705
C09702=1046.007,67.581,-83.342,170.306,35.631,156.705
C09703=1046.014,67.830,-83.360,170.307,35.632,156.705
C09704=1046.020,68.078,-83.378,170.309,35.633,156.705
C09705=1046.026,68.328,-83.396,170.311,35.635,156.706
C09706=1046.032,68.578,-83.414,170.312,35.637,156.706
C09707=1046.038,68.827,-83.432,170.314,35.638,156.706
C09708=1046.045,69.076,-83.449,170.316,35.640,156.707
C09709=1046.051,69.326,-83.467,170.317,35.641,156.707
C09710=1046.057,69.575,-83.486,170.320,35.643,156.707
C09711=1046.063,69.824,-83.504,170.322,35.644,156.707
C09712=1046.069,70.073,-83.522,170.323,35.646,156.708
C09713=1046.076,70.322,-83.540,170.325,35.647,156.708
C09714=1046.082,70.572,-83.558,170.326,35.649,156.708
C09715=1046.088,70.821,-83.576,170.328,35.651,156.709
C09716=1046.094,71.070,-83.594,170.330,35.652,156.709
C09717=1046.100,71.319,-83.612,170.331,35.654,156.709
C09718=1046.107,71.569,-83.630,170.334,35.655,156.709
C09719=1046.113,71.818,-83.649,170.336,35.657,156.710
C09720=1046.118,72.067,-83.667,170.337,35.658,156.710
C09721=1046.125,72.317,-83.684,170.339,35.660,156.710
C09722=1046.132,72.566,-83.703,170.341,35.661,156.711
C09723=1046.138,72.816,-83.720,170.342,35.663,156.711
C09724=1046.144,73.065,-83.739,170.344,35.665,156.711
C09725=1046.150,73.314,-83.757,170.345,35.666,156.711
C09726=1046.156,73.563,-83.775,170.348,35.668,156.712
C09727=1046.162,73.813,-83.793,170.350,35.669,156.712
C09728=1046.169,74.062,-83.812,170.351,35.670,156.712
C09729=1046.175,74.311,-83.831,170.353,35.672,156.712
C09730=1046.181,74.560,-83.848,170.355,35.674,156.713
C09731=1046.187,74.809,-83.867,170.356,35.675,156.713
C09732=1046.193,75.059,-83.885,170.358,35.677,156.713
C09733=1046.200,75.308,-83.903,170.360,35.678,156.713
C09734=1046.206,75.558,-83.921,170.362,35.680,156.714
C09735=1046.212,75.807,-83.940,170.364,35.681,156.714
C09736=1046.218,76.056,-83.957,170.366,35.683,156.714
C09737=1046.224,76.305,-83.976,170.367,35.684,156.715
C09738=1046.231,76.554,-83.994,170.369,35.686,156.715
C09739=1046.237,76.803,-84.012,170.371,35.688,156.715
C09740=1046.244,77.089,-84.033,170.372,35.690,156.716
C09741=1046.252,77.375,-84.054,170.375,35.691,156.716
C09742=1046.259,77.661,-84.076,170.377,35.693,156.716
C09743=1046.266,77.947,-84.097,170.379,35.695,156.716
C09744=1046.272,78.197,-84.115,170.381,35.697,156.717
C09745=1046.278,78.446,-84.134,170.382,35.698,156.717
C09746=1046.285,78.695,-84.153,170.384,35.700,156.717
C09747=1046.290,78.944,-84.170,170.386,35.701,156.718
C09748=1046.296,79.193,-84.189,170.387,35.703,156.718
C09749=1046.303,79.442,-84.207,170.390,35.704,156.718
C09750=1046.309,79.692,-84.227,170.392,35.706,156.719
C09751=1046.315,79.941,-84.245,170.393,35.707,156.719
C09752=1046.321,80.191,-84.263,170.395,35.709,156.719
C09753=1046.328,80.440,-84.282,170.396,35.711,156.719
C09754=1046.333,80.688,-84.300,170.398,35.712,156.720
C09755=1046.340,80.938,-84.318,170.400,35.714,156.720
C09756=1046.345,81.187,-84.337,170.402,35.716,156.720
C09757=1046.352,81.436,-84.356,170.404,35.717,156.720
C09758=1046.358,81.685,-84.375,170.406,35.719,156.721
C09759=1046.364,81.935,-84.393,170.407,35.720,156.721
C09760=1046.370,82.185,-84.412,170.409,35.722,156.721
C09761=1046.376,82.434,-84.430,170.410,35.723,156.722
C09762=1046.383,82.683,-84.449,170.412,35.725,156.722
C09763=1046.389,82.932,-84.468,170.414,35.726,156.722
C09764=1046.395,83.180,-84.486,170.416,35.728,156.723
C09765=1046.401,83.430,-84.505,170.418,35.730,156.723
C09766=1046.407,83.680,-84.523,170.420,35.732,156.723
C09767=1046.413,83.929,-84.542,170.421,35.733,156.723
C09768=1046.420,84.178,-84.561,170.423,35.735,156.724
C09769=1046.426,84.427,-84.579,170.425,35.736,156.724
C09770=1046.432,84.676,-84.598,170.426,35.738,156.724
C09771=1046.438,84.926,-84.617,170.429,35.739,156.724
C09772=1046.445,85.175,-84.636,170.431,35.741,156.725
C09773=1046.451,85.424,-84.654,170.432,35.742,156.725
C09774=1046.457,85.673,-84.674,170.434,35.744,156.725
C09775=1046.463,85.922,-84.692,170.436,35.745,156.726
C09776=1046.470,86.171,-84.711,170.437,35.747,156.726
C09777=1046.476,86.421,-84.729,170.439,35.749,156.726
C09778=1046.481,86.671,-84.748,170.441,35.751,156.727
C09779=1046.488,86.920,-84.767,170.443,35.752,156.727
C09780=1046.494,87.169,-84.785,170.445,35.754,156.727
C09781=1046.501,87.418,-84.804,170.446,35.755,156.727
C09782=1046.507,87.667,-84.823,170.448,35.756,156.728
C09783=1046.513,87.917,-84.842,170.450,35.758,156.728
C09784=1046.519,88.166,-84.861,170.451,35.759,156.728
C09785=1046.526,88.415,-84.879,170.453,35.761,156.728
C09786=1046.532,88.664,-84.898,170.456,35.763,156.729
C09787=1046.538,88.913,-84.917,170.457,35.765,156.729
C09788=1046.544,89.162,-84.936,170.459,35.766,156.729
C09789=1046.551,89.412,-84.954,170.461,35.768,156.730
C09790=1046.556,89.661,-84.974,170.462,35.769,156.730
C09791=1046.563,89.910,-84.992,170.464,35.771,156.730
C09792=1046.569,90.159,-85.012,170.466,35.772,156.730
C09793=1046.576,90.408,-85.030,170.467,35.773,156.731
C09794=1046.582,90.657,-85.050,170.470,35.775,156.731
C09795=1046.588,90.906,-85.068,170.472,35.777,156.731
C09796=1046.594,91.156,-85.087,170.473,35.778,156.732
C09797=1046.600,91.405,-85.106,170.475,35.780,156.732
C09798=1046.606,91.654,-85.125,170.477,35.782,156.732
C09799=1046.612,91.903,-85.144,170.478,35.784,156.733
C09800=1046.618,92.152,-85.164,170.481,35.785,156.733
C09801=1046.624,92.402,-85.183,170.482,35.787,156.733
C09802=1046.630,92.651,-85.202,170.484,35.789,156.733
C09803=1046.636,92.900,-85.221,170.486,35.790,156.734
C09804=1046.643,93.186,-85.243,170.488,35.792,156.734
C09805=1046.651,93.472,-85.265,170.489,35.794,156.734
C09806=1046.658,93.759,-85.287,170.491,35.796,156.735
C09807=1046.665,94.044,-85.309,170.494,35.797,156.735
C09808=1046.670,94.293,-85.328,170.496,35.799,156.735
C09809=1046.677,94.543,-85.347,170.498,35.801,156.736
C09810=1046.683,94.792,-85.367,170.499,35.803,156.736
C09811=1046.690,95.041,-85.386,170.501,35.804,156.736
C09812=1046.695,95.290,-85.405,170.503,35.806,156.737
C09813=1046.702,95.539,-85.423,170.504,35.807,156.737
C09814=1046.708,95.788,-85.443,170.507,35.809,156.737
C09815=1046.714,96.037,-85.462,170.509,35.811,156.737
C09816=1046.720,96.287,-85.481,170.510,35.812,156.738
C09817=1046.727,96.535,-85.501,170.512,35.814,156.738
C09818=1046.732,96.785,-85.520,170.513,35.815,156.738
C09819=1046.739,97.034,-85.539,170.515,35.817,156.739
C09820=1046.745,97.283,-85.559,170.517,35.818,156.739
C09821=1046.751,97.533,-85.578,170.519,35.820,156.739
C09822=1046.757,97.782,-85.597,170.521,35.821,156.739
C09823=1046.763,98.031,-85.617,170.523,35.823,156.740
C09824=1046.770,98.280,-85.635,170.524,35.825,156.740
C09825=1046.776,98.529,-85.655,170.526,35.827,156.740
C09826=1046.782,98.778,-85.674,170.528,35.828,156.741
C09827=1046.789,99.028,-85.694,170.529,35.830,156.741
C09828=1046.794,99.277,-85.713,170.532,35.832,156.741
C09829=1046.801,99.526,-85.732,170.534,35.833,156.742
C09830=1046.807,99.775,-85.751,170.535,35.835,156.742
C09831=1046.813,100.024,-85.771,170.537,35.836,156.742
C09832=1046.819,100.273,-85.790,170.539,35.838,156.742
C09833=1046.826,100.523,-85.809,170.541,35.839,156.743
C09834=1046.832,100.772,-85.829,170.542,35.841,156.743
C09835=1046.838,101.021,-85.848,170.545,35.843,156.743
C09836=1046.844,101.270,-85.868,170.546,35.844,156.744
C09837=1046.849,101.519,-85.887,170.548,35.846,156.744
C09838=1046.856,101.768,-85.907,170.550,35.847,156.744
C09839=1046.862,102.017,-85.926,170.551,35.849,156.745
C09840=1046.868,102.267,-85.946,170.553,35.851,156.745
C09841=1046.874,102.516,-85.966,170.555,35.852,156.745
C09842=1046.880,102.765,-85.986,170.557,35.854,156.745
C09843=1046.887,103.014,-86.004,170.559,35.856,156.746
C09844=1046.893,103.263,-86.024,170.561,35.857,156.746
C09845=1046.899,103.512,-86.044,170.562,35.859,156.746
C09846=1046.905,103.762,-86.064,170.564,35.861,156.747
C09847=1046.911,104.011,-86.084,170.566,35.863,156.747
C09848=1046.917,104.260,-86.103,170.568,35.864,156.747
C09849=1046.923,104.509,-86.122,170.570,35.866,156.748
C09850=1046.929,104.758,-86.142,170.572,35.868,156.748
C09851=1046.936,105.008,-86.162,170.573,35.869,156.748
C09852=1046.942,105.257,-86.182,170.575,35.871,156.749
C09853=1046.947,105.506,-86.201,170.577,35.873,156.749
C09854=1046.953,105.755,-86.221,170.578,35.874,156.749
C09855=1046.961,106.004,-86.241,170.581,35.876,156.749
C09856=1046.966,106.253,-86.260,170.583,35.878,156.750
C09857=1046.972,106.502,-86.280,170.584,35.880,156.750
C09858=1046.978,106.751,-86.300,170.586,35.881,156.750
C09859=1046.984,107.000,-86.319,170.588,35.883,156.751
C09860=1046.991,107.250,-86.339,170.589,35.884,156.751
C09861=1046.997,107.498,-86.359,170.592,35.886,156.751
C09862=1047.003,107.748,-86.378,170.594,35.888,156.752
C09863=1047.010,107.997,-86.398,170.596,35.889,156.752
C09864=1047.016,108.246,-86.418,170.597,35.891,156.752
C09865=1047.021,108.496,-86.438,170.599,35.892,156.752
C09866=1047.027,108.744,-86.458,170.601,35.894,156.753
C09867=1047.034,108.994,-86.478,170.602,35.896,156.753
C09868=1047.041,109.280,-86.500,170.605,35.898,156.754
C09869=1047.048,109.566,-86.523,170.607,35.900,156.754
C09870=1047.055,109.851,-86.546,170.609,35.902,156.754
C09871=1047.062,110.137,-86.568,170.611,35.903,156.755
C09872=1047.068,110.386,-86.588,170.613,35.905,156.755
C09873=1047.075,110.635,-86.608,170.614,35.907,156.755
C09874=1047.081,110.885,-86.627,170.617,35.908,156.755
C09875=1047.087,111.134,-86.647,170.619,35.910,156.756
C09876=1047.093,111.383,-86.667,170.620,35.912,156.756
C09877=1047.100,111.632,-86.688,170.622,35.913,156.756
C09878=1047.106,111.881,-86.708,170.624,35.915,156.757
C09879=1047.112,112.130,-86.728,170.626,35.917,156.757
C09880=1047.118,112.380,-86.747,170.627,35.918,156.757
C09881=1047.124,112.629,-86.767,170.630,35.920,156.758
C09882=1047.130,112.877,-86.787,170.632,35.922,156.758
C09883=1047.137,113.127,-86.807,170.633,35.923,156.758
C09884=1047.143,113.376,-86.827,170.635,35.925,156.759
C09885=1047.148,113.625,-86.848,170.637,35.927,156.759
C09886=1047.154,113.874,-86.868,170.638,35.928,156.759
C09887=1047.160,114.123,-86.888,170.641,35.930,156.759
C09888=1047.166,114.372,-86.908,170.643,35.932,156.760
C09889=1047.172,114.621,-86.928,170.644,35.934,156.760
C09890=1047.178,114.871,-86.949,170.646,35.935,156.760
C09891=1047.184,115.119,-86.969,170.648,35.937,156.761
C09892=1047.190,115.368,-86.989,170.649,35.939,156.761
C09893=1047.196,115.618,-87.010,170.652,35.940,156.761
C09894=1047.202,115.867,-87.030,170.654,35.942,156.762
C09895=1047.208,116.116,-87.050,170.656,35.944,156.762
C09896=1047.215,116.365,-87.070,170.657,35.946,156.762
C09897=1047.220,116.614,-87.091,170.659,35.947,156.763
C09898=1047.226,116.863,-87.111,170.661,35.949,156.763
C09899=1047.233,117.113,-87.131,170.663,35.951,156.763
C09900=1047.239,117.362,-87.151,170.665,35.952,156.764
C09901=1047.244,117.611,-87.171,170.667,35.954,156.764
C09902=1047.250,117.860,-87.192,170.668,35.956,156.764
C09903=1047.256,118.109,-87.212,170.670,35.958,156.765
C09904=1047.262,118.358,-87.232,170.672,35.959,156.765
C09905=1047.268,118.608,-87.253,170.674,35.961,156.765
C09906=1047.275,118.856,-87.273,170.676,35.963,156.766
C09907=1047.281,119.105,-87.294,170.678,35.965,156.766
C09908=1047.286,119.354,-87.314,170.680,35.966,156.766
C09909=1047.292,119.603,-87.334,170.681,35.968,156.767
C09910=1047.299,119.853,-87.354,170.683,35.970,156.767
C09911=1047.304,120.102,-87.375,170.686,35.972,156.767
C09912=1047.311,120.351,-87.395,170.687,35.973,156.768
C09913=1047.317,120.600,-87.416,170.689,35.975,156.768
C09914=1047.322,120.849,-87.437,170.691,35.977,156.768
C09915=1047.329,121.098,-87.457,170.693,35.979,156.769
C09916=1047.335,121.347,-87.477,170.694,35.980,156.769
C09917=1047.341,121.597,-87.498,170.697,35.982,156.769
C09918=1047.347,121.845,-87.518,170.699,35.984,156.770
C09919=1047.353,122.094,-87.538,170.700,35.986,156.770
C09920=1047.359,122.344,-87.559,170.702,35.987,156.770
C09921=1047.365,122.593,-87.579,170.704,35.989,156.770
C09922=1047.372,122.842,-87.600,170.706,35.991,156.771
C09923=1047.378,123.090,-87.620,170.708,35.992,156.771
C09924=1047.384,123.340,-87.641,170.710,35.994,156.771
C09925=1047.390,123.589,-87.661,170.712,35.996,156.772
C09926=1047.396,123.838,-87.682,170.713,35.997,156.772
C09927=1047.402,124.087,-87.703,170.715,35.999,156.772
C09928=1047.408,124.336,-87.723,170.717,36.001,156.773
C09929=1047.414,124.585,-87.743,170.720,36.003,156.773
C09930=1047.421,124.834,-87.765,170.721,36.004,156.773
C09931=1047.427,125.083,-87.785,170.723,36.006,156.774
C09932=1047.434,125.369,-87.808,170.725,36.008,156.774
C09933=1047.441,125.655,-87.832,170.727,36.010,156.774
C09934=1047.448,125.941,-87.855,170.729,36.012,156.775
C09935=1047.455,126.226,-87.879,170.732,36.014,156.775
C09936=1047.461,126.476,-87.900,170.734,36.016,156.776
C09937=1047.467,126.724,-87.921,170.736,36.017,156.776
C09938=1047.474,126.974,-87.941,170.737,36.019,156.776
C09939=1047.479,127.222,-87.962,170.739,36.021,156.776
C09940=1047.486,127.472,-87.982,170.741,36.023,156.777
C09941=1047.492,127.722,-88.003,170.744,36.024,156.777
C09942=1047.498,127.970,-88.024,170.745,36.026,156.777
C09943=1047.505,128.219,-88.044,170.747,36.028,156.778
C09944=1047.510,128.468,-88.066,170.749,36.029,156.778
C09945=1047.517,128.717,-88.086,170.751,36.031,156.778
C09946=1047.523,128.966,-88.106,170.753,36.033,156.779
C09947=1047.529,129.215,-88.128,170.755,36.034,156.779
C09948=1047.535,129.465,-88.148,170.757,36.036,156.779
C09949=1047.542,129.713,-88.169,170.759,36.038,156.780
C09950=1047.548,129.963,-88.189,170.761,36.039,156.780
C09951=1047.554,130.211,-88.210,170.762,36.041,156.780
C09952=1047.560,130.461,-88.231,170.764,36.042,156.781
C09953=1047.567,130.710,-88.252,170.767,36.044,156.781
C09954=1047.573,130.959,-88.272,170.769,36.046,156.781
C09955=1047.579,131.208,-88.294,170.771,36.048,156.782
C09956=1047.585,131.457,-88.314,170.772,36.049,156.782
C09957=1047.591,131.706,-88.335,170.774,36.051,156.782
C09958=1047.597,131.956,-88.356,170.776,36.053,156.783
C09959=1047.603,132.204,-88.377,170.779,36.054,156.783
C09960=1047.609,132.453,-88.399,170.780,36.056,156.783
C09961=1047.615,132.702,-88.419,170.782,36.058,156.784
C09962=1047.621,132.951,-88.440,170.784,36.060,156.784
C09963=1047.627,133.201,-88.461,170.786,36.062,156.784
C09964=1047.633,133.449,-88.482,170.788,36.064,156.785
C09965=1047.640,133.698,-88.503,170.790,36.066,156.785
C09966=1047.645,133.947,-88.524,170.792,36.067,156.785
C09967=1047.651,134.197,-88.546,170.794,36.069,156.786
C09968=1047.658,134.445,-88.567,170.795,36.071,156.786
C09969=1047.663,134.695,-88.587,170.797,36.072,156.786
C09970=1047.670,134.944,-88.609,170.800,36.074,156.787
C09971=1047.676,135.192,-88.629,170.802,36.076,156.787
C09972=1047.682,135.441,-88.651,170.804,36.077,156.787
C09973=1047.688,135.691,-88.672,170.805,36.079,156.788
C09974=1047.694,135.939,-88.693,170.807,36.081,156.788
C09975=1047.700,136.188,-88.714,170.809,36.083,156.788
C09976=1047.706,136.438,-88.735,170.812,36.085,156.789
C09977=1047.712,136.686,-88.756,170.814,36.087,156.789
C09978=1047.719,136.936,-88.778,170.815,36.088,156.789
C09979=1047.725,137.185,-88.799,170.817,36.090,156.790
C09980=1047.730,137.433,-88.820,170.819,36.092,156.790
C09981=1047.737,137.683,-88.841,170.822,36.094,156.790
C09982=1047.743,137.932,-88.862,170.823,36.095,156.791
C09983=1047.749,138.181,-88.884,170.825,36.097,156.791
C09984=1047.755,138.430,-88.905,170.827,36.099,156.791
C09985=1047.762,138.679,-88.926,170.829,36.101,156.792
C09986=1047.767,138.928,-88.947,170.831,36.102,156.792
C09987=1047.773,139.177,-88.969,170.833,36.104,156.792
C09988=1047.779,139.426,-88.990,170.835,36.106,156.793
C09989=1047.785,139.675,-89.012,170.837,36.108,156.793
C09990=1047.792,139.924,-89.032,170.839,36.110,156.793
C09991=1047.798,140.173,-89.054,170.841,36.112,156.794
C09992=1047.804,140.422,-89.076,170.843,36.113,156.794
C09993=1047.810,140.670,-89.097,170.845,36.115,156.794
C09994=1047.816,140.920,-89.119,170.847,36.117,156.795
C09995=1047.822,141.169,-89.140,170.849,36.119,156.795
C09996=1047.828,141.455,-89.165,170.851,36.121,156.796
//INST
///DATE 2021/06/17 10:57
///ATTR SC,RW,RJ
////FRAME ROBOT
///GROUP1 RB1
NOP
MOVL C00000 V=800.0 PL=0
MOVL C00001 V=800.0 PL=0
MOVL C00002 V=800.0 PL=0
MOVL C00003 V=800.0 PL=0
MOVL C00004 V=800.0 PL=0
MOVL C00005 V=800.0 PL=0
MOVL C00006 V=800.0 PL=0
MOVL C00007 V=800.0 PL=0
MOVL C00008 V=800.0 PL=0
MOVL C00009 V=800.0 PL=0
MOVL C00010 V=800.0 PL=0
MOVL C00011 V=800.0 PL=0
MOVL C00012 V=800.0 PL=0
MOVL C00013 V=800.0 PL=0
MOVL C00014 V=800.0 PL=0
MOVL C00015 V=800.0 PL=0
MOVL C00016 V=800.0 PL=0
MOVL C00017 V=800.0 PL=0
MOVL C00018 V=800.0 PL=0
MOVL C00019 V=800.0 PL=0
MOVL C00020 V=800.0 PL=0
MOVL C00021 V=800.0 PL=0
MOVL C00022 V=800.0 PL=0
MOVL C00023 V=800.0 PL=0
MOVL C00024 V=800.0 PL=0
MOVL C00025 V=800.0 PL=0
MOVL C00026 V=800.0 PL=0
MOVL C00027 V=800.0 PL=0
MOVL C00028 V=800.0 PL=0
MOVL C00029 V=800.0 PL=0
MOVL C00030 V=800.0 PL=0
MOVL C00031 V=800.0 PL=0
MOVL C00032 V=800.0 PL=0
MOVL C00033 V=800.0 PL=0
MOVL C00034 V=800.0 PL=0
MOVL C00035 V=800.0 PL=0
MOVL C00036 V=800.0 PL=0
MOVL C00037 V=800.0 PL=0
MOVL C00038 V=800.0 PL=0
MOVL C00039 V=800.0 PL=0
MOVL C00040 V=800.0 PL=0
MOVL C00041 V=800.0 PL=0
MOVL C00042 V=800.0 PL=0
MOVL C00043 V=800.0 PL=0
MOVL C00044 V=800.0 PL=0
MOVL C00045 V=800.0 PL=0
MOVL C00046 V=800.0 PL=0
MOVL C00047 V=800.0 PL=0
MOVL C00048 V=800.0 PL=0
MOVL C00049 V=800.0 PL=0
MOVL C00050 V=800.0 PL=0
MOVL C00051 V=800.0 PL=0
MOVL C00052 V=800.0 PL=0
MOVL C00053 V=800.0 PL=0
MOVL C00054 V=800.0 PL=0
MOVL C00055 V=800.0 PL=0
MOVL C00056 V=800.0 PL=0
MOVL C00057 V=800.0 PL=0
MOVL C00058 V=800.0 PL=0
MOVL C00059 V=800.0 PL=0
MOVL C00060 V=800.0 PL=0
MOVL C00061 V=800.0 PL=0
MOVL C00062 V=800.0 PL=0
MOVL C00063 V=800.0 PL=0
MOVL C00064 V=800.0 PL=0
MOVL C00065 V=800.0 PL=0
MOVL C00066 V=800.0 PL=0
MOVL C00067 V=800.0 PL=0
MOVL C00068 V=800.0 PL=0
MOVL C00069 V=800.0 PL=0
MOVL C00070 V=800.0 PL=0
MOVL C00071 V=800.0 PL=0
MOVL C00072 V=800.0 PL=0
MOVL C00073 V=800.0 PL=0
MOVL C00074 V=800.0 PL=0
MOVL C00075 V=800.0 PL=0
MOVL C00076 V=800.0 PL=0
MOVL C00077 V=800.0 PL=0
MOVL C00078 V=800.0 PL=0
MOVL C00079 V=800.0 PL=0
MOVL C00080 V=800.0 PL=0
MOVL C00081 V=800.0 PL=0
MOVL C00082 V=800.0 PL=0
MOVL C00083 V=800.0 PL=0
MOVL C00084 V=800.0 PL=0
MOVL C00085 V=800.0 PL=0
MOVL C00086 V=800.0 PL=0
MOVL C00087 V=800.0 PL=0
MOVL C00088 V=800.0 PL=0
MOVL C00089 V=800.0 PL=0
MOVL C00090 V=800.0 PL=0
MOVL C00091 V=800.0 PL=0
MOVL C00092 V=800.0 PL=0
MOVL C00093 V=800.0 PL=0
MOVL C00094 V=800.0 PL=0
MOVL C00095 V=800.0 PL=0
MOVL C00096 V=800.0 PL=0
MOVL C00097 V=800.0 PL=0
MOVL C00098 V=800.0 PL=0
MOVL C00099 V=800.0 PL=0
MOVL C00100 V=800.0 PL=0
MOVL C00101 V=800.0 PL=0
MOVL C00102 V=800.0 PL=0
MOVL C00103 V=800.0 PL=0
MOVL C00104 V=800.0 PL=0
MOVL C00105 V=800.0 PL=0
MOVL C00106 V=800.0 PL=0
MOVL C00107 V=800.0 PL=0
MOVL C00108 V=800.0 PL=0
MOVL C00109 V=800.0 PL=0
MOVL C00110 V=800.0 PL=0
MOVL C00111 V=800.0 PL=0
MOVL C00112 V=800.0 PL=0
MOVL C00113 V=800.0 PL=0
MOVL C00114 V=800.0 PL=0
MOVL C00115 V=800.0 PL=0
MOVL C00116 V=800.0 PL=0
MOVL C00117 V=800.0 PL=0
MOVL C00118 V=800.0 PL=0
MOVL C00119 V=800.0 PL=0
MOVL C00120 V=800.0 PL=0
MOVL C00121 V=800.0 PL=0
MOVL C00122 V=800.0 PL=0
MOVL C00123 V=800.0 PL=0
MOVL C00124 V=800.0 PL=0
MOVL C00125 V=800.0 PL=0
MOVL C00126 V=800.0 PL=0
MOVL C00127 V=800.0 PL=0
MOVL C00128 V=800.0 PL=0
MOVL C00129 V=800.0 PL=0
MOVL C00130 V=800.0 PL=0
MOVL C00131 V=800.0 PL=0
MOVL C00132 V=800.0 PL=0
MOVL C00133 V=800.0 PL=0
MOVL C00134 V=800.0 PL=0
MOVL C00135 V=800.0 PL=0
MOVL C00136 V=800.0 PL=0
MOVL C00137 V=800.0 PL=0
MOVL C00138 V=800.0 PL=0
MOVL C00139 V=800.0 PL=0
MOVL C00140 V=800.0 PL=0
MOVL C00141 V=800.0 PL=0
MOVL C00142 V=800.0 PL=0
MOVL C00143 V=800.0 PL=0
MOVL C00144 V=800.0 PL=0
MOVL C00145 V=800.0 PL=0
MOVL C00146 V=800.0 PL=0
MOVL C00147 V=800.0 PL=0
MOVL C00148 V=800.0 PL=0
MOVL C00149 V=800.0 PL=0
MOVL C00150 V=800.0 PL=0
MOVL C00151 V=800.0 PL=0
MOVL C00152 V=800.0 PL=0
MOVL C00153 V=800.0 PL=0
MOVL C00154 V=800.0 PL=0
MOVL C00155 V=800.0 PL=0
MOVL C00156 V=800.0 PL=0
MOVL C00157 V=800.0 PL=0
MOVL C00158 V=800.0 PL=0
MOVL C00159 V=800.0 PL=0
MOVL C00160 V=800.0 PL=0
MOVL C00161 V=800.0 PL=0
MOVL C00162 V=800.0 PL=0
MOVL C00163 V=800.0 PL=0
MOVL C00164 V=800.0 PL=0
MOVL C00165 V=800.0 PL=0
MOVL C00166 V=800.0 PL=0
MOVL C00167 V=800.0 PL=0
MOVL C00168 V=800.0 PL=0
MOVL C00169 V=800.0 PL=0
MOVL C00170 V=800.0 PL=0
MOVL C00171 V=800.0 PL=0
MOVL C00172 V=800.0 PL=0
MOVL C00173 V=800.0 PL=0
MOVL C00174 V=800.0 PL=0
MOVL C00175 V=800.0 PL=0
MOVL C00176 V=800.0 PL=0
MOVL C00177 V=800.0 PL=0
MOVL C00178 V=800.0 PL=0
MOVL C00179 V=800.0 PL=0
MOVL C00180 V=800.0 PL=0
MOVL C00181 V=800.0 PL=0
MOVL C00182 V=800.0 PL=0
MOVL C00183 V=800.0 PL=0
MOVL C00184 V=800.0 PL=0
MOVL C00185 V=800.0 PL=0
MOVL C00186 V=800.0 PL=0
MOVL C00187 V=800.0 PL=0
MOVL C00188 V=800.0 PL=0
MOVL C00189 V=800.0 PL=0
MOVL C00190 V=800.0 PL=0
MOVL C00191 V=800.0 PL=0
MOVL C00192 V=800.0 PL=0
MOVL C00193 V=800.0 PL=0
MOVL C00194 V=800.0 PL=0
MOVL C00195 V=800.0 PL=0
MOVL C00196 V=800.0 PL=0
MOVL C00197 V=800.0 PL=0
MOVL C00198 V=800.0 PL=0
MOVL C00199 V=800.0 PL=0
MOVL C00200 V=800.0 PL=0
MOVL C00201 V=800.0 PL=0
MOVL C00202 V=800.0 PL=0
MOVL C00203 V=800.0 PL=0
MOVL C00204 V=800.0 PL=0
MOVL C00205 V=800.0 PL=0
MOVL C00206 V=800.0 PL=0
MOVL C00207 V=800.0 PL=0
MOVL C00208 V=800.0 PL=0
MOVL C00209 V=800.0 PL=0
MOVL C00210 V=800.0 PL=0
MOVL C00211 V=800.0 PL=0
MOVL C00212 V=800.0 PL=0
MOVL C00213 V=800.0 PL=0
MOVL C00214 V=800.0 PL=0
MOVL C00215 V=800.0 PL=0
MOVL C00216 V=800.0 PL=0
MOVL C00217 V=800.0 PL=0
MOVL C00218 V=800.0 PL=0
MOVL C00219 V=800.0 PL=0
MOVL C00220 V=800.0 PL=0
MOVL C00221 V=800.0 PL=0
MOVL C00222 V=800.0 PL=0
MOVL C00223 V=800.0 PL=0
MOVL C00224 V=800.0 PL=0
MOVL C00225 V=800.0 PL=0
MOVL C00226 V=800.0 PL=0
MOVL C00227 V=800.0 PL=0
MOVL C00228 V=800.0 PL=0
MOVL C00229 V=800.0 PL=0
MOVL C00230 V=800.0 PL=0
MOVL C00231 V=800.0 PL=0
MOVL C00232 V=800.0 PL=0
MOVL C00233 V=800.0 PL=0
MOVL C00234 V=800.0 PL=0
MOVL C00235 V=800.0 PL=0
MOVL C00236 V=800.0 PL=0
MOVL C00237 V=800.0 PL=0
MOVL C00238 V=800.0 PL=0
MOVL C00239 V=800.0 PL=0
MOVL C00240 V=800.0 PL=0
MOVL C00241 V=800.0 PL=0
MOVL C00242 V=800.0 PL=0
MOVL C00243 V=800.0 PL=0
MOVL C00244 V=800.0 PL=0
MOVL C00245 V=800.0 PL=0
MOVL C00246 V=800.0 PL=0
MOVL C00247 V=800.0 PL=0
MOVL C00248 V=800.0 PL=0
MOVL C00249 V=800.0 PL=0
MOVL C00250 V=800.0 PL=0
MOVL C00251 V=800.0 PL=0
MOVL C00252 V=800.0 PL=0
MOVL C00253 V=800.0 PL=0
MOVL C00254 V=800.0 PL=0
MOVL C00255 V=800.0 PL=0
MOVL C00256 V=800.0 PL=0
MOVL C00257 V=800.0 PL=0
MOVL C00258 V=800.0 PL=0
MOVL C00259 V=800.0 PL=0
MOVL C00260 V=800.0 PL=0
MOVL C00261 V=800.0 PL=0
MOVL C00262 V=800.0 PL=0
MOVL C00263 V=800.0 PL=0
MOVL C00264 V=800.0 PL=0
MOVL C00265 V=800.0 PL=0
MOVL C00266 V=800.0 PL=0
MOVL C00267 V=800.0 PL=0
MOVL C00268 V=800.0 PL=0
MOVL C00269 V=800.0 PL=0
MOVL C00270 V=800.0 PL=0
MOVL C00271 V=800.0 PL=0
MOVL C00272 V=800.0 PL=0
MOVL C00273 V=800.0 PL=0
MOVL C00274 V=800.0 PL=0
MOVL C00275 V=800.0 PL=0
MOVL C00276 V=800.0 PL=0
MOVL C00277 V=800.0 PL=0
MOVL C00278 V=800.0 PL=0
MOVL C00279 V=800.0 PL=0
MOVL C00280 V=800.0 PL=0
MOVL C00281 V=800.0 PL=0
MOVL C00282 V=800.0 PL=0
MOVL C00283 V=800.0 PL=0
MOVL C00284 V=800.0 PL=0
MOVL C00285 V=800.0 PL=0
MOVL C00286 V=800.0 PL=0
MOVL C00287 V=800.0 PL=0
MOVL C00288 V=800.0 PL=0
MOVL C00289 V=800.0 PL=0
MOVL C00290 V=800.0 PL=0
MOVL C00291 V=800.0 PL=0
MOVL C00292 V=800.0 PL=0
MOVL C00293 V=800.0 PL=0
MOVL C00294 V=800.0 PL=0
MOVL C00295 V=800.0 PL=0
MOVL C00296 V=800.0 PL=0
MOVL C00297 V=800.0 PL=0
MOVL C00298 V=800.0 PL=0
MOVL C00299 V=800.0 PL=0
MOVL C00300 V=800.0 PL=0
MOVL C00301 V=800.0 PL=0
MOVL C00302 V=800.0 PL=0
MOVL C00303 V=800.0 PL=0
MOVL C00304 V=800.0 PL=0
MOVL C00305 V=800.0 PL=0
MOVL C00306 V=800.0 PL=0
MOVL C00307 V=800.0 PL=0
MOVL C00308 V=800.0 PL=0
MOVL C00309 V=800.0 PL=0
MOVL C00310 V=800.0 PL=0
MOVL C00311 V=800.0 PL=0
MOVL C00312 V=800.0 PL=0
MOVL C00313 V=800.0 PL=0
MOVL C00314 V=800.0 PL=0
MOVL C00315 V=800.0 PL=0
MOVL C00316 V=800.0 PL=0
MOVL C00317 V=800.0 PL=0
MOVL C00318 V=800.0 PL=0
MOVL C00319 V=800.0 PL=0
MOVL C00320 V=800.0 PL=0
MOVL C00321 V=800.0 PL=0
MOVL C00322 V=800.0 PL=0
MOVL C00323 V=800.0 PL=0
MOVL C00324 V=800.0 PL=0
MOVL C00325 V=800.0 PL=0
MOVL C00326 V=800.0 PL=0
MOVL C00327 V=800.0 PL=0
MOVL C00328 V=800.0 PL=0
MOVL C00329 V=800.0 PL=0
MOVL C00330 V=800.0 PL=0
MOVL C00331 V=800.0 PL=0
MOVL C00332 V=800.0 PL=0
MOVL C00333 V=800.0 PL=0
MOVL C00334 V=800.0 PL=0
MOVL C00335 V=800.0 PL=0
MOVL C00336 V=800.0 PL=0
MOVL C00337 V=800.0 PL=0
MOVL C00338 V=800.0 PL=0
MOVL C00339 V=800.0 PL=0
MOVL C00340 V=800.0 PL=0
MOVL C00341 V=800.0 PL=0
MOVL C00342 V=800.0 PL=0
MOVL C00343 V=800.0 PL=0
MOVL C00344 V=800.0 PL=0
MOVL C00345 V=800.0 PL=0
MOVL C00346 V=800.0 PL=0
MOVL C00347 V=800.0 PL=0
MOVL C00348 V=800.0 PL=0
MOVL C00349 V=800.0 PL=0
MOVL C00350 V=800.0 PL=0
MOVL C00351 V=800.0 PL=0
MOVL C00352 V=800.0 PL=0
MOVL C00353 V=800.0 PL=0
MOVL C00354 V=800.0 PL=0
MOVL C00355 V=800.0 PL=0
MOVL C00356 V=800.0 PL=0
MOVL C00357 V=800.0 PL=0
MOVL C00358 V=800.0 PL=0
MOVL C00359 V=800.0 PL=0
MOVL C00360 V=800.0 PL=0
MOVL C00361 V=800.0 PL=0
MOVL C00362 V=800.0 PL=0
MOVL C00363 V=800.0 PL=0
MOVL C00364 V=800.0 PL=0
MOVL C00365 V=800.0 PL=0
MOVL C00366 V=800.0 PL=0
MOVL C00367 V=800.0 PL=0
MOVL C00368 V=800.0 PL=0
MOVL C00369 V=800.0 PL=0
MOVL C00370 V=800.0 PL=0
MOVL C00371 V=800.0 PL=0
MOVL C00372 V=800.0 PL=0
MOVL C00373 V=800.0 PL=0
MOVL C00374 V=800.0 PL=0
MOVL C00375 V=800.0 PL=0
MOVL C00376 V=800.0 PL=0
MOVL C00377 V=800.0 PL=0
MOVL C00378 V=800.0 PL=0
MOVL C00379 V=800.0 PL=0
MOVL C00380 V=800.0 PL=0
MOVL C00381 V=800.0 PL=0
MOVL C00382 V=800.0 PL=0
MOVL C00383 V=800.0 PL=0
MOVL C00384 V=800.0 PL=0
MOVL C00385 V=800.0 PL=0
MOVL C00386 V=800.0 PL=0
MOVL C00387 V=800.0 PL=0
MOVL C00388 V=800.0 PL=0
MOVL C00389 V=800.0 PL=0
MOVL C00390 V=800.0 PL=0
MOVL C00391 V=800.0 PL=0
MOVL C00392 V=800.0 PL=0
MOVL C00393 V=800.0 PL=0
MOVL C00394 V=800.0 PL=0
MOVL C00395 V=800.0 PL=0
MOVL C00396 V=800.0 PL=0
MOVL C00397 V=800.0 PL=0
MOVL C00398 V=800.0 PL=0
MOVL C00399 V=800.0 PL=0
MOVL C00400 V=800.0 PL=0
MOVL C00401 V=800.0 PL=0
MOVL C00402 V=800.0 PL=0
MOVL C00403 V=800.0 PL=0
MOVL C00404 V=800.0 PL=0
MOVL C00405 V=800.0 PL=0
MOVL C00406 V=800.0 PL=0
MOVL C00407 V=800.0 PL=0
MOVL C00408 V=800.0 PL=0
MOVL C00409 V=800.0 PL=0
MOVL C00410 V=800.0 PL=0
MOVL C00411 V=800.0 PL=0
MOVL C00412 V=800.0 PL=0
MOVL C00413 V=800.0 PL=0
MOVL C00414 V=800.0 PL=0
MOVL C00415 V=800.0 PL=0
MOVL C00416 V=800.0 PL=0
MOVL C00417 V=800.0 PL=0
MOVL C00418 V=800.0 PL=0
MOVL C00419 V=800.0 PL=0
MOVL C00420 V=800.0 PL=0
MOVL C00421 V=800.0 PL=0
MOVL C00422 V=800.0 PL=0
MOVL C00423 V=800.0 PL=0
MOVL C00424 V=800.0 PL=0
MOVL C00425 V=800.0 PL=0
MOVL C00426 V=800.0 PL=0
MOVL C00427 V=800.0 PL=0
MOVL C00428 V=800.0 PL=0
MOVL C00429 V=800.0 PL=0
MOVL C00430 V=800.0 PL=0
MOVL C00431 V=800.0 PL=0
MOVL C00432 V=800.0 PL=0
MOVL C00433 V=800.0 PL=0
MOVL C00434 V=800.0 PL=0
MOVL C00435 V=800.0 PL=0
MOVL C00436 V=800.0 PL=0
MOVL C00437 V=800.0 PL=0
MOVL C00438 V=800.0 PL=0
MOVL C00439 V=800.0 PL=0
MOVL C00440 V=800.0 PL=0
MOVL C00441 V=800.0 PL=0
MOVL C00442 V=800.0 PL=0
MOVL C00443 V=800.0 PL=0
MOVL C00444 V=800.0 PL=0
MOVL C00445 V=800.0 PL=0
MOVL C00446 V=800.0 PL=0
MOVL C00447 V=800.0 PL=0
MOVL C00448 V=800.0 PL=0
MOVL C00449 V=800.0 PL=0
MOVL C00450 V=800.0 PL=0
MOVL C00451 V=800.0 PL=0
MOVL C00452 V=800.0 PL=0
MOVL C00453 V=800.0 PL=0
MOVL C00454 V=800.0 PL=0
MOVL C00455 V=800.0 PL=0
MOVL C00456 V=800.0 PL=0
MOVL C00457 V=800.0 PL=0
MOVL C00458 V=800.0 PL=0
MOVL C00459 V=800.0 PL=0
MOVL C00460 V=800.0 PL=0
MOVL C00461 V=800.0 PL=0
MOVL C00462 V=800.0 PL=0
MOVL C00463 V=800.0 PL=0
MOVL C00464 V=800.0 PL=0
MOVL C00465 V=800.0 PL=0
MOVL C00466 V=800.0 PL=0
MOVL C00467 V=800.0 PL=0
MOVL C00468 V=800.0 PL=0
MOVL C00469 V=800.0 PL=0
MOVL C00470 V=800.0 PL=0
MOVL C00471 V=800.0 PL=0
MOVL C00472 V=800.0 PL=0
MOVL C00473 V=800.0 PL=0
MOVL C00474 V=800.0 PL=0
MOVL C00475 V=800.0 PL=0
MOVL C00476 V=800.0 PL=0
MOVL C00477 V=800.0 PL=0
MOVL C00478 V=800.0 PL=0
MOVL C00479 V=800.0 PL=0
MOVL C00480 V=800.0 PL=0
MOVL C00481 V=800.0 PL=0
MOVL C00482 V=800.0 PL=0
MOVL C00483 V=800.0 PL=0
MOVL C00484 V=800.0 PL=0
MOVL C00485 V=800.0 PL=0
MOVL C00486 V=800.0 PL=0
MOVL C00487 V=800.0 PL=0
MOVL C00488 V=800.0 PL=0
MOVL C00489 V=800.0 PL=0
MOVL C00490 V=800.0 PL=0
MOVL C00491 V=800.0 PL=0
MOVL C00492 V=800.0 PL=0
MOVL C00493 V=800.0 PL=0
MOVL C00494 V=800.0 PL=0
MOVL C00495 V=800.0 PL=0
MOVL C00496 V=800.0 PL=0
MOVL C00497 V=800.0 PL=0
MOVL C00498 V=800.0 PL=0
MOVL C00499 V=800.0 PL=0
MOVL C00500 V=800.0 PL=0
MOVL C00501 V=800.0 PL=0
MOVL C00502 V=800.0 PL=0
MOVL C00503 V=800.0 PL=0
MOVL C00504 V=800.0 PL=0
MOVL C00505 V=800.0 PL=0
MOVL C00506 V=800.0 PL=0
MOVL C00507 V=800.0 PL=0
MOVL C00508 V=800.0 PL=0
MOVL C00509 V=800.0 PL=0
MOVL C00510 V=800.0 PL=0
MOVL C00511 V=800.0 PL=0
MOVL C00512 V=800.0 PL=0
MOVL C00513 V=800.0 PL=0
MOVL C00514 V=800.0 PL=0
MOVL C00515 V=800.0 PL=0
MOVL C00516 V=800.0 PL=0
MOVL C00517 V=800.0 PL=0
MOVL C00518 V=800.0 PL=0
MOVL C00519 V=800.0 PL=0
MOVL C00520 V=800.0 PL=0
MOVL C00521 V=800.0 PL=0
MOVL C00522 V=800.0 PL=0
MOVL C00523 V=800.0 PL=0
MOVL C00524 V=800.0 PL=0
MOVL C00525 V=800.0 PL=0
MOVL C00526 V=800.0 PL=0
MOVL C00527 V=800.0 PL=0
MOVL C00528 V=800.0 PL=0
MOVL C00529 V=800.0 PL=0
MOVL C00530 V=800.0 PL=0
MOVL C00531 V=800.0 PL=0
MOVL C00532 V=800.0 PL=0
MOVL C00533 V=800.0 PL=0
MOVL C00534 V=800.0 PL=0
MOVL C00535 V=800.0 PL=0
MOVL C00536 V=800.0 PL=0
MOVL C00537 V=800.0 PL=0
MOVL C00538 V=800.0 PL=0
MOVL C00539 V=800.0 PL=0
MOVL C00540 V=800.0 PL=0
MOVL C00541 V=800.0 PL=0
MOVL C00542 V=800.0 PL=0
MOVL C00543 V=800.0 PL=0
MOVL C00544 V=800.0 PL=0
MOVL C00545 V=800.0 PL=0
MOVL C00546 V=800.0 PL=0
MOVL C00547 V=800.0 PL=0
MOVL C00548 V=800.0 PL=0
MOVL C00549 V=800.0 PL=0
MOVL C00550 V=800.0 PL=0
MOVL C00551 V=800.0 PL=0
MOVL C00552 V=800.0 PL=0
MOVL C00553 V=800.0 PL=0
MOVL C00554 V=800.0 PL=0
MOVL C00555 V=800.0 PL=0
MOVL C00556 V=800.0 PL=0
MOVL C00557 V=800.0 PL=0
MOVL C00558 V=800.0 PL=0
MOVL C00559 V=800.0 PL=0
MOVL C00560 V=800.0 PL=0
MOVL C00561 V=800.0 PL=0
MOVL C00562 V=800.0 PL=0
MOVL C00563 V=800.0 PL=0
MOVL C00564 V=800.0 PL=0
MOVL C00565 V=800.0 PL=0
MOVL C00566 V=800.0 PL=0
MOVL C00567 V=800.0 PL=0
MOVL C00568 V=800.0 PL=0
MOVL C00569 V=800.0 PL=0
MOVL C00570 V=800.0 PL=0
MOVL C00571 V=800.0 PL=0
MOVL C00572 V=800.0 PL=0
MOVL C00573 V=800.0 PL=0
MOVL C00574 V=800.0 PL=0
MOVL C00575 V=800.0 PL=0
MOVL C00576 V=800.0 PL=0
MOVL C00577 V=800.0 PL=0
MOVL C00578 V=800.0 PL=0
MOVL C00579 V=800.0 PL=0
MOVL C00580 V=800.0 PL=0
MOVL C00581 V=800.0 PL=0
MOVL C00582 V=800.0 PL=0
MOVL C00583 V=800.0 PL=0
MOVL C00584 V=800.0 PL=0
MOVL C00585 V=800.0 PL=0
MOVL C00586 V=800.0 PL=0
MOVL C00587 V=800.0 PL=0
MOVL C00588 V=800.0 PL=0
MOVL C00589 V=800.0 PL=0
MOVL C00590 V=800.0 PL=0
MOVL C00591 V=800.0 PL=0
MOVL C00592 V=800.0 PL=0
MOVL C00593 V=800.0 PL=0
MOVL C00594 V=800.0 PL=0
MOVL C00595 V=800.0 PL=0
MOVL C00596 V=800.0 PL=0
MOVL C00597 V=800.0 PL=0
MOVL C00598 V=800.0 PL=0
MOVL C00599 V=800.0 PL=0
MOVL C00600 V=800.0 PL=0
MOVL C00601 V=800.0 PL=0
MOVL C00602 V=800.0 PL=0
MOVL C00603 V=800.0 PL=0
MOVL C00604 V=800.0 PL=0
MOVL C00605 V=800.0 PL=0
MOVL C00606 V=800.0 PL=0
MOVL C00607 V=800.0 PL=0
MOVL C00608 V=800.0 PL=0
MOVL C00609 V=800.0 PL=0
MOVL C00610 V=800.0 PL=0
MOVL C00611 V=800.0 PL=0
MOVL C00612 V=800.0 PL=0
MOVL C00613 V=800.0 PL=0
MOVL C00614 V=800.0 PL=0
MOVL C00615 V=800.0 PL=0
MOVL C00616 V=800.0 PL=0
MOVL C00617 V=800.0 PL=0
MOVL C00618 V=800.0 PL=0
MOVL C00619 V=800.0 PL=0
MOVL C00620 V=800.0 PL=0
MOVL C00621 V=800.0 PL=0
MOVL C00622 V=800.0 PL=0
MOVL C00623 V=800.0 PL=0
MOVL C00624 V=800.0 PL=0
MOVL C00625 V=800.0 PL=0
MOVL C00626 V=800.0 PL=0
MOVL C00627 V=800.0 PL=0
MOVL C00628 V=800.0 PL=0
MOVL C00629 V=800.0 PL=0
MOVL C00630 V=800.0 PL=0
MOVL C00631 V=800.0 PL=0
MOVL C00632 V=800.0 PL=0
MOVL C00633 V=800.0 PL=0
MOVL C00634 V=800.0 PL=0
MOVL C00635 V=800.0 PL=0
MOVL C00636 V=800.0 PL=0
MOVL C00637 V=800.0 PL=0
MOVL C00638 V=800.0 PL=0
MOVL C00639 V=800.0 PL=0
MOVL C00640 V=800.0 PL=0
MOVL C00641 V=800.0 PL=0
MOVL C00642 V=800.0 PL=0
MOVL C00643 V=800.0 PL=0
MOVL C00644 V=800.0 PL=0
MOVL C00645 V=800.0 PL=0
MOVL C00646 V=800.0 PL=0
MOVL C00647 V=800.0 PL=0
MOVL C00648 V=800.0 PL=0
MOVL C00649 V=800.0 PL=0
MOVL C00650 V=800.0 PL=0
MOVL C00651 V=800.0 PL=0
MOVL C00652 V=800.0 PL=0
MOVL C00653 V=800.0 PL=0
MOVL C00654 V=800.0 PL=0
MOVL C00655 V=800.0 PL=0
MOVL C00656 V=800.0 PL=0
MOVL C00657 V=800.0 PL=0
MOVL C00658 V=800.0 PL=0
MOVL C00659 V=800.0 PL=0
MOVL C00660 V=800.0 PL=0
MOVL C00661 V=800.0 PL=0
MOVL C00662 V=800.0 PL=0
MOVL C00663 V=800.0 PL=0
MOVL C00664 V=800.0 PL=0
MOVL C00665 V=800.0 PL=0
MOVL C00666 V=800.0 PL=0
MOVL C00667 V=800.0 PL=0
MOVL C00668 V=800.0 PL=0
MOVL C00669 V=800.0 PL=0
MOVL C00670 V=800.0 PL=0
MOVL C00671 V=800.0 PL=0
MOVL C00672 V=800.0 PL=0
MOVL C00673 V=800.0 PL=0
MOVL C00674 V=800.0 PL=0
MOVL C00675 V=800.0 PL=0
MOVL C00676 V=800.0 PL=0
MOVL C00677 V=800.0 PL=0
MOVL C00678 V=800.0 PL=0
MOVL C00679 V=800.0 PL=0
MOVL C00680 V=800.0 PL=0
MOVL C00681 V=800.0 PL=0
MOVL C00682 V=800.0 PL=0
MOVL C00683 V=800.0 PL=0
MOVL C00684 V=800.0 PL=0
MOVL C00685 V=800.0 PL=0
MOVL C00686 V=800.0 PL=0
MOVL C00687 V=800.0 PL=0
MOVL C00688 V=800.0 PL=0
MOVL C00689 V=800.0 PL=0
MOVL C00690 V=800.0 PL=0
MOVL C00691 V=800.0 PL=0
MOVL C00692 V=800.0 PL=0
MOVL C00693 V=800.0 PL=0
MOVL C00694 V=800.0 PL=0
MOVL C00695 V=800.0 PL=0
MOVL C00696 V=800.0 PL=0
MOVL C00697 V=800.0 PL=0
MOVL C00698 V=800.0 PL=0
MOVL C00699 V=800.0 PL=0
MOVL C00700 V=800.0 PL=0
MOVL C00701 V=800.0 PL=0
MOVL C00702 V=800.0 PL=0
MOVL C00703 V=800.0 PL=0
MOVL C00704 V=800.0 PL=0
MOVL C00705 V=800.0 PL=0
MOVL C00706 V=800.0 PL=0
MOVL C00707 V=800.0 PL=0
MOVL C00708 V=800.0 PL=0
MOVL C00709 V=800.0 PL=0
MOVL C00710 V=800.0 PL=0
MOVL C00711 V=800.0 PL=0
MOVL C00712 V=800.0 PL=0
MOVL C00713 V=800.0 PL=0
MOVL C00714 V=800.0 PL=0
MOVL C00715 V=800.0 PL=0
MOVL C00716 V=800.0 PL=0
MOVL C00717 V=800.0 PL=0
MOVL C00718 V=800.0 PL=0
MOVL C00719 V=800.0 PL=0
MOVL C00720 V=800.0 PL=0
MOVL C00721 V=800.0 PL=0
MOVL C00722 V=800.0 PL=0
MOVL C00723 V=800.0 PL=0
MOVL C00724 V=800.0 PL=0
MOVL C00725 V=800.0 PL=0
MOVL C00726 V=800.0 PL=0
MOVL C00727 V=800.0 PL=0
MOVL C00728 V=800.0 PL=0
MOVL C00729 V=800.0 PL=0
MOVL C00730 V=800.0 PL=0
MOVL C00731 V=800.0 PL=0
MOVL C00732 V=800.0 PL=0
MOVL C00733 V=800.0 PL=0
MOVL C00734 V=800.0 PL=0
MOVL C00735 V=800.0 PL=0
MOVL C00736 V=800.0 PL=0
MOVL C00737 V=800.0 PL=0
MOVL C00738 V=800.0 PL=0
MOVL C00739 V=800.0 PL=0
MOVL C00740 V=800.0 PL=0
MOVL C00741 V=800.0 PL=0
MOVL C00742 V=800.0 PL=0
MOVL C00743 V=800.0 PL=0
MOVL C00744 V=800.0 PL=0
MOVL C00745 V=800.0 PL=0
MOVL C00746 V=800.0 PL=0
MOVL C00747 V=800.0 PL=0
MOVL C00748 V=800.0 PL=0
MOVL C00749 V=800.0 PL=0
MOVL C00750 V=800.0 PL=0
MOVL C00751 V=800.0 PL=0
MOVL C00752 V=800.0 PL=0
MOVL C00753 V=800.0 PL=0
MOVL C00754 V=800.0 PL=0
MOVL C00755 V=800.0 PL=0
MOVL C00756 V=800.0 PL=0
MOVL C00757 V=800.0 PL=0
MOVL C00758 V=800.0 PL=0
MOVL C00759 V=800.0 PL=0
MOVL C00760 V=800.0 PL=0
MOVL C00761 V=800.0 PL=0
MOVL C00762 V=800.0 PL=0
MOVL C00763 V=800.0 PL=0
MOVL C00764 V=800.0 PL=0
MOVL C00765 V=800.0 PL=0
MOVL C00766 V=800.0 PL=0
MOVL C00767 V=800.0 PL=0
MOVL C00768 V=800.0 PL=0
MOVL C00769 V=800.0 PL=0
MOVL C00770 V=800.0 PL=0
MOVL C00771 V=800.0 PL=0
MOVL C00772 V=800.0 PL=0
MOVL C00773 V=800.0 PL=0
MOVL C00774 V=800.0 PL=0
MOVL C00775 V=800.0 PL=0
MOVL C00776 V=800.0 PL=0
MOVL C00777 V=800.0 PL=0
MOVL C00778 V=800.0 PL=0
MOVL C00779 V=800.0 PL=0
MOVL C00780 V=800.0 PL=0
MOVL C00781 V=800.0 PL=0
MOVL C00782 V=800.0 PL=0
MOVL C00783 V=800.0 PL=0
MOVL C00784 V=800.0 PL=0
MOVL C00785 V=800.0 PL=0
MOVL C00786 V=800.0 PL=0
MOVL C00787 V=800.0 PL=0
MOVL C00788 V=800.0 PL=0
MOVL C00789 V=800.0 PL=0
MOVL C00790 V=800.0 PL=0
MOVL C00791 V=800.0 PL=0
MOVL C00792 V=800.0 PL=0
MOVL C00793 V=800.0 PL=0
MOVL C00794 V=800.0 PL=0
MOVL C00795 V=800.0 PL=0
MOVL C00796 V=800.0 PL=0
MOVL C00797 V=800.0 PL=0
MOVL C00798 V=800.0 PL=0
MOVL C00799 V=800.0 PL=0
MOVL C00800 V=800.0 PL=0
MOVL C00801 V=800.0 PL=0
MOVL C00802 V=800.0 PL=0
MOVL C00803 V=800.0 PL=0
MOVL C00804 V=800.0 PL=0
MOVL C00805 V=800.0 PL=0
MOVL C00806 V=800.0 PL=0
MOVL C00807 V=800.0 PL=0
MOVL C00808 V=800.0 PL=0
MOVL C00809 V=800.0 PL=0
MOVL C00810 V=800.0 PL=0
MOVL C00811 V=800.0 PL=0
MOVL C00812 V=800.0 PL=0
MOVL C00813 V=800.0 PL=0
MOVL C00814 V=800.0 PL=0
MOVL C00815 V=800.0 PL=0
MOVL C00816 V=800.0 PL=0
MOVL C00817 V=800.0 PL=0
MOVL C00818 V=800.0 PL=0
MOVL C00819 V=800.0 PL=0
MOVL C00820 V=800.0 PL=0
MOVL C00821 V=800.0 PL=0
MOVL C00822 V=800.0 PL=0
MOVL C00823 V=800.0 PL=0
MOVL C00824 V=800.0 PL=0
MOVL C00825 V=800.0 PL=0
MOVL C00826 V=800.0 PL=0
MOVL C00827 V=800.0 PL=0
MOVL C00828 V=800.0 PL=0
MOVL C00829 V=800.0 PL=0
MOVL C00830 V=800.0 PL=0
MOVL C00831 V=800.0 PL=0
MOVL C00832 V=800.0 PL=0
MOVL C00833 V=800.0 PL=0
MOVL C00834 V=800.0 PL=0
MOVL C00835 V=800.0 PL=0
MOVL C00836 V=800.0 PL=0
MOVL C00837 V=800.0 PL=0
MOVL C00838 V=800.0 PL=0
MOVL C00839 V=800.0 PL=0
MOVL C00840 V=800.0 PL=0
MOVL C00841 V=800.0 PL=0
MOVL C00842 V=800.0 PL=0
MOVL C00843 V=800.0 PL=0
MOVL C00844 V=800.0 PL=0
MOVL C00845 V=800.0 PL=0
MOVL C00846 V=800.0 PL=0
MOVL C00847 V=800.0 PL=0
MOVL C00848 V=800.0 PL=0
MOVL C00849 V=800.0 PL=0
MOVL C00850 V=800.0 PL=0
MOVL C00851 V=800.0 PL=0
MOVL C00852 V=800.0 PL=0
MOVL C00853 V=800.0 PL=0
MOVL C00854 V=800.0 PL=0
MOVL C00855 V=800.0 PL=0
MOVL C00856 V=800.0 PL=0
MOVL C00857 V=800.0 PL=0
MOVL C00858 V=800.0 PL=0
MOVL C00859 V=800.0 PL=0
MOVL C00860 V=800.0 PL=0
MOVL C00861 V=800.0 PL=0
MOVL C00862 V=800.0 PL=0
MOVL C00863 V=800.0 PL=0
MOVL C00864 V=800.0 PL=0
MOVL C00865 V=800.0 PL=0
MOVL C00866 V=800.0 PL=0
MOVL C00867 V=800.0 PL=0
MOVL C00868 V=800.0 PL=0
MOVL C00869 V=800.0 PL=0
MOVL C00870 V=800.0 PL=0
MOVL C00871 V=800.0 PL=0
MOVL C00872 V=800.0 PL=0
MOVL C00873 V=800.0 PL=0
MOVL C00874 V=800.0 PL=0
MOVL C00875 V=800.0 PL=0
MOVL C00876 V=800.0 PL=0
MOVL C00877 V=800.0 PL=0
MOVL C00878 V=800.0 PL=0
MOVL C00879 V=800.0 PL=0
MOVL C00880 V=800.0 PL=0
MOVL C00881 V=800.0 PL=0
MOVL C00882 V=800.0 PL=0
MOVL C00883 V=800.0 PL=0
MOVL C00884 V=800.0 PL=0
MOVL C00885 V=800.0 PL=0
MOVL C00886 V=800.0 PL=0
MOVL C00887 V=800.0 PL=0
MOVL C00888 V=800.0 PL=0
MOVL C00889 V=800.0 PL=0
MOVL C00890 V=800.0 PL=0
MOVL C00891 V=800.0 PL=0
MOVL C00892 V=800.0 PL=0
MOVL C00893 V=800.0 PL=0
MOVL C00894 V=800.0 PL=0
MOVL C00895 V=800.0 PL=0
MOVL C00896 V=800.0 PL=0
MOVL C00897 V=800.0 PL=0
MOVL C00898 V=800.0 PL=0
MOVL C00899 V=800.0 PL=0
MOVL C00900 V=800.0 PL=0
MOVL C00901 V=800.0 PL=0
MOVL C00902 V=800.0 PL=0
MOVL C00903 V=800.0 PL=0
MOVL C00904 V=800.0 PL=0
MOVL C00905 V=800.0 PL=0
MOVL C00906 V=800.0 PL=0
MOVL C00907 V=800.0 PL=0
MOVL C00908 V=800.0 PL=0
MOVL C00909 V=800.0 PL=0
MOVL C00910 V=800.0 PL=0
MOVL C00911 V=800.0 PL=0
MOVL C00912 V=800.0 PL=0
MOVL C00913 V=800.0 PL=0
MOVL C00914 V=800.0 PL=0
MOVL C00915 V=800.0 PL=0
MOVL C00916 V=800.0 PL=0
MOVL C00917 V=800.0 PL=0
MOVL C00918 V=800.0 PL=0
MOVL C00919 V=800.0 PL=0
MOVL C00920 V=800.0 PL=0
MOVL C00921 V=800.0 PL=0
MOVL C00922 V=800.0 PL=0
MOVL C00923 V=800.0 PL=0
MOVL C00924 V=800.0 PL=0
MOVL C00925 V=800.0 PL=0
MOVL C00926 V=800.0 PL=0
MOVL C00927 V=800.0 PL=0
MOVL C00928 V=800.0 PL=0
MOVL C00929 V=800.0 PL=0
MOVL C00930 V=800.0 PL=0
MOVL C00931 V=800.0 PL=0
MOVL C00932 V=800.0 PL=0
MOVL C00933 V=800.0 PL=0
MOVL C00934 V=800.0 PL=0
MOVL C00935 V=800.0 PL=0
MOVL C00936 V=800.0 PL=0
MOVL C00937 V=800.0 PL=0
MOVL C00938 V=800.0 PL=0
MOVL C00939 V=800.0 PL=0
MOVL C00940 V=800.0 PL=0
MOVL C00941 V=800.0 PL=0
MOVL C00942 V=800.0 PL=0
MOVL C00943 V=800.0 PL=0
MOVL C00944 V=800.0 PL=0
MOVL C00945 V=800.0 PL=0
MOVL C00946 V=800.0 PL=0
MOVL C00947 V=800.0 PL=0
MOVL C00948 V=800.0 PL=0
MOVL C00949 V=800.0 PL=0
MOVL C00950 V=800.0 PL=0
MOVL C00951 V=800.0 PL=0
MOVL C00952 V=800.0 PL=0
MOVL C00953 V=800.0 PL=0
MOVL C00954 V=800.0 PL=0
MOVL C00955 V=800.0 PL=0
MOVL C00956 V=800.0 PL=0
MOVL C00957 V=800.0 PL=0
MOVL C00958 V=800.0 PL=0
MOVL C00959 V=800.0 PL=0
MOVL C00960 V=800.0 PL=0
MOVL C00961 V=800.0 PL=0
MOVL C00962 V=800.0 PL=0
MOVL C00963 V=800.0 PL=0
MOVL C00964 V=800.0 PL=0
MOVL C00965 V=800.0 PL=0
MOVL C00966 V=800.0 PL=0
MOVL C00967 V=800.0 PL=0
MOVL C00968 V=800.0 PL=0
MOVL C00969 V=800.0 PL=0
MOVL C00970 V=800.0 PL=0
MOVL C00971 V=800.0 PL=0
MOVL C00972 V=800.0 PL=0
MOVL C00973 V=800.0 PL=0
MOVL C00974 V=800.0 PL=0
MOVL C00975 V=800.0 PL=0
MOVL C00976 V=800.0 PL=0
MOVL C00977 V=800.0 PL=0
MOVL C00978 V=800.0 PL=0
MOVL C00979 V=800.0 PL=0
MOVL C00980 V=800.0 PL=0
MOVL C00981 V=800.0 PL=0
MOVL C00982 V=800.0 PL=0
MOVL C00983 V=800.0 PL=0
MOVL C00984 V=800.0 PL=0
MOVL C00985 V=800.0 PL=0
MOVL C00986 V=800.0 PL=0
MOVL C00987 V=800.0 PL=0
MOVL C00988 V=800.0 PL=0
MOVL C00989 V=800.0 PL=0
MOVL C00990 V=800.0 PL=0
MOVL C00991 V=800.0 PL=0
MOVL C00992 V=800.0 PL=0
MOVL C00993 V=800.0 PL=0
MOVL C00994 V=800.0 PL=0
MOVL C00995 V=800.0 PL=0
MOVL C00996 V=800.0 PL=0
MOVL C00997 V=800.0 PL=0
MOVL C00998 V=800.0 PL=0
MOVL C00999 V=800.0 PL=0
MOVL C01000 V=800.0 PL=0
MOVL C01001 V=800.0 PL=0
MOVL C01002 V=800.0 PL=0
MOVL C01003 V=800.0 PL=0
MOVL C01004 V=800.0 PL=0
MOVL C01005 V=800.0 PL=0
MOVL C01006 V=800.0 PL=0
MOVL C01007 V=800.0 PL=0
MOVL C01008 V=800.0 PL=0
MOVL C01009 V=800.0 PL=0
MOVL C01010 V=800.0 PL=0
MOVL C01011 V=800.0 PL=0
MOVL C01012 V=800.0 PL=0
MOVL C01013 V=800.0 PL=0
MOVL C01014 V=800.0 PL=0
MOVL C01015 V=800.0 PL=0
MOVL C01016 V=800.0 PL=0
MOVL C01017 V=800.0 PL=0
MOVL C01018 V=800.0 PL=0
MOVL C01019 V=800.0 PL=0
MOVL C01020 V=800.0 PL=0
MOVL C01021 V=800.0 PL=0
MOVL C01022 V=800.0 PL=0
MOVL C01023 V=800.0 PL=0
MOVL C01024 V=800.0 PL=0
MOVL C01025 V=800.0 PL=0
MOVL C01026 V=800.0 PL=0
MOVL C01027 V=800.0 PL=0
MOVL C01028 V=800.0 PL=0
MOVL C01029 V=800.0 PL=0
MOVL C01030 V=800.0 PL=0
MOVL C01031 V=800.0 PL=0
MOVL C01032 V=800.0 PL=0
MOVL C01033 V=800.0 PL=0
MOVL C01034 V=800.0 PL=0
MOVL C01035 V=800.0 PL=0
MOVL C01036 V=800.0 PL=0
MOVL C01037 V=800.0 PL=0
MOVL C01038 V=800.0 PL=0
MOVL C01039 V=800.0 PL=0
MOVL C01040 V=800.0 PL=0
MOVL C01041 V=800.0 PL=0
MOVL C01042 V=800.0 PL=0
MOVL C01043 V=800.0 PL=0
MOVL C01044 V=800.0 PL=0
MOVL C01045 V=800.0 PL=0
MOVL C01046 V=800.0 PL=0
MOVL C01047 V=800.0 PL=0
MOVL C01048 V=800.0 PL=0
MOVL C01049 V=800.0 PL=0
MOVL C01050 V=800.0 PL=0
MOVL C01051 V=800.0 PL=0
MOVL C01052 V=800.0 PL=0
MOVL C01053 V=800.0 PL=0
MOVL C01054 V=800.0 PL=0
MOVL C01055 V=800.0 PL=0
MOVL C01056 V=800.0 PL=0
MOVL C01057 V=800.0 PL=0
MOVL C01058 V=800.0 PL=0
MOVL C01059 V=800.0 PL=0
MOVL C01060 V=800.0 PL=0
MOVL C01061 V=800.0 PL=0
MOVL C01062 V=800.0 PL=0
MOVL C01063 V=800.0 PL=0
MOVL C01064 V=800.0 PL=0
MOVL C01065 V=800.0 PL=0
MOVL C01066 V=800.0 PL=0
MOVL C01067 V=800.0 PL=0
MOVL C01068 V=800.0 PL=0
MOVL C01069 V=800.0 PL=0
MOVL C01070 V=800.0 PL=0
MOVL C01071 V=800.0 PL=0
MOVL C01072 V=800.0 PL=0
MOVL C01073 V=800.0 PL=0
MOVL C01074 V=800.0 PL=0
MOVL C01075 V=800.0 PL=0
MOVL C01076 V=800.0 PL=0
MOVL C01077 V=800.0 PL=0
MOVL C01078 V=800.0 PL=0
MOVL C01079 V=800.0 PL=0
MOVL C01080 V=800.0 PL=0
MOVL C01081 V=800.0 PL=0
MOVL C01082 V=800.0 PL=0
MOVL C01083 V=800.0 PL=0
MOVL C01084 V=800.0 PL=0
MOVL C01085 V=800.0 PL=0
MOVL C01086 V=800.0 PL=0
MOVL C01087 V=800.0 PL=0
MOVL C01088 V=800.0 PL=0
MOVL C01089 V=800.0 PL=0
MOVL C01090 V=800.0 PL=0
MOVL C01091 V=800.0 PL=0
MOVL C01092 V=800.0 PL=0
MOVL C01093 V=800.0 PL=0
MOVL C01094 V=800.0 PL=0
MOVL C01095 V=800.0 PL=0
MOVL C01096 V=800.0 PL=0
MOVL C01097 V=800.0 PL=0
MOVL C01098 V=800.0 PL=0
MOVL C01099 V=800.0 PL=0
MOVL C01100 V=800.0 PL=0
MOVL C01101 V=800.0 PL=0
MOVL C01102 V=800.0 PL=0
MOVL C01103 V=800.0 PL=0
MOVL C01104 V=800.0 PL=0
MOVL C01105 V=800.0 PL=0
MOVL C01106 V=800.0 PL=0
MOVL C01107 V=800.0 PL=0
MOVL C01108 V=800.0 PL=0
MOVL C01109 V=800.0 PL=0
MOVL C01110 V=800.0 PL=0
MOVL C01111 V=800.0 PL=0
MOVL C01112 V=800.0 PL=0
MOVL C01113 V=800.0 PL=0
MOVL C01114 V=800.0 PL=0
MOVL C01115 V=800.0 PL=0
MOVL C01116 V=800.0 PL=0
MOVL C01117 V=800.0 PL=0
MOVL C01118 V=800.0 PL=0
MOVL C01119 V=800.0 PL=0
MOVL C01120 V=800.0 PL=0
MOVL C01121 V=800.0 PL=0
MOVL C01122 V=800.0 PL=0
MOVL C01123 V=800.0 PL=0
MOVL C01124 V=800.0 PL=0
MOVL C01125 V=800.0 PL=0
MOVL C01126 V=800.0 PL=0
MOVL C01127 V=800.0 PL=0
MOVL C01128 V=800.0 PL=0
MOVL C01129 V=800.0 PL=0
MOVL C01130 V=800.0 PL=0
MOVL C01131 V=800.0 PL=0
MOVL C01132 V=800.0 PL=0
MOVL C01133 V=800.0 PL=0
MOVL C01134 V=800.0 PL=0
MOVL C01135 V=800.0 PL=0
MOVL C01136 V=800.0 PL=0
MOVL C01137 V=800.0 PL=0
MOVL C01138 V=800.0 PL=0
MOVL C01139 V=800.0 PL=0
MOVL C01140 V=800.0 PL=0
MOVL C01141 V=800.0 PL=0
MOVL C01142 V=800.0 PL=0
MOVL C01143 V=800.0 PL=0
MOVL C01144 V=800.0 PL=0
MOVL C01145 V=800.0 PL=0
MOVL C01146 V=800.0 PL=0
MOVL C01147 V=800.0 PL=0
MOVL C01148 V=800.0 PL=0
MOVL C01149 V=800.0 PL=0
MOVL C01150 V=800.0 PL=0
MOVL C01151 V=800.0 PL=0
MOVL C01152 V=800.0 PL=0
MOVL C01153 V=800.0 PL=0
MOVL C01154 V=800.0 PL=0
MOVL C01155 V=800.0 PL=0
MOVL C01156 V=800.0 PL=0
MOVL C01157 V=800.0 PL=0
MOVL C01158 V=800.0 PL=0
MOVL C01159 V=800.0 PL=0
MOVL C01160 V=800.0 PL=0
MOVL C01161 V=800.0 PL=0
MOVL C01162 V=800.0 PL=0
MOVL C01163 V=800.0 PL=0
MOVL C01164 V=800.0 PL=0
MOVL C01165 V=800.0 PL=0
MOVL C01166 V=800.0 PL=0
MOVL C01167 V=800.0 PL=0
MOVL C01168 V=800.0 PL=0
MOVL C01169 V=800.0 PL=0
MOVL C01170 V=800.0 PL=0
MOVL C01171 V=800.0 PL=0
MOVL C01172 V=800.0 PL=0
MOVL C01173 V=800.0 PL=0
MOVL C01174 V=800.0 PL=0
MOVL C01175 V=800.0 PL=0
MOVL C01176 V=800.0 PL=0
MOVL C01177 V=800.0 PL=0
MOVL C01178 V=800.0 PL=0
MOVL C01179 V=800.0 PL=0
MOVL C01180 V=800.0 PL=0
MOVL C01181 V=800.0 PL=0
MOVL C01182 V=800.0 PL=0
MOVL C01183 V=800.0 PL=0
MOVL C01184 V=800.0 PL=0
MOVL C01185 V=800.0 PL=0
MOVL C01186 V=800.0 PL=0
MOVL C01187 V=800.0 PL=0
MOVL C01188 V=800.0 PL=0
MOVL C01189 V=800.0 PL=0
MOVL C01190 V=800.0 PL=0
MOVL C01191 V=800.0 PL=0
MOVL C01192 V=800.0 PL=0
MOVL C01193 V=800.0 PL=0
MOVL C01194 V=800.0 PL=0
MOVL C01195 V=800.0 PL=0
MOVL C01196 V=800.0 PL=0
MOVL C01197 V=800.0 PL=0
MOVL C01198 V=800.0 PL=0
MOVL C01199 V=800.0 PL=0
MOVL C01200 V=800.0 PL=0
MOVL C01201 V=800.0 PL=0
MOVL C01202 V=800.0 PL=0
MOVL C01203 V=800.0 PL=0
MOVL C01204 V=800.0 PL=0
MOVL C01205 V=800.0 PL=0
MOVL C01206 V=800.0 PL=0
MOVL C01207 V=800.0 PL=0
MOVL C01208 V=800.0 PL=0
MOVL C01209 V=800.0 PL=0
MOVL C01210 V=800.0 PL=0
MOVL C01211 V=800.0 PL=0
MOVL C01212 V=800.0 PL=0
MOVL C01213 V=800.0 PL=0
MOVL C01214 V=800.0 PL=0
MOVL C01215 V=800.0 PL=0
MOVL C01216 V=800.0 PL=0
MOVL C01217 V=800.0 PL=0
MOVL C01218 V=800.0 PL=0
MOVL C01219 V=800.0 PL=0
MOVL C01220 V=800.0 PL=0
MOVL C01221 V=800.0 PL=0
MOVL C01222 V=800.0 PL=0
MOVL C01223 V=800.0 PL=0
MOVL C01224 V=800.0 PL=0
MOVL C01225 V=800.0 PL=0
MOVL C01226 V=800.0 PL=0
MOVL C01227 V=800.0 PL=0
MOVL C01228 V=800.0 PL=0
MOVL C01229 V=800.0 PL=0
MOVL C01230 V=800.0 PL=0
MOVL C01231 V=800.0 PL=0
MOVL C01232 V=800.0 PL=0
MOVL C01233 V=800.0 PL=0
MOVL C01234 V=800.0 PL=0
MOVL C01235 V=800.0 PL=0
MOVL C01236 V=800.0 PL=0
MOVL C01237 V=800.0 PL=0
MOVL C01238 V=800.0 PL=0
MOVL C01239 V=800.0 PL=0
MOVL C01240 V=800.0 PL=0
MOVL C01241 V=800.0 PL=0
MOVL C01242 V=800.0 PL=0
MOVL C01243 V=800.0 PL=0
MOVL C01244 V=800.0 PL=0
MOVL C01245 V=800.0 PL=0
MOVL C01246 V=800.0 PL=0
MOVL C01247 V=800.0 PL=0
MOVL C01248 V=800.0 PL=0
MOVL C01249 V=800.0 PL=0
MOVL C01250 V=800.0 PL=0
MOVL C01251 V=800.0 PL=0
MOVL C01252 V=800.0 PL=0
MOVL C01253 V=800.0 PL=0
MOVL C01254 V=800.0 PL=0
MOVL C01255 V=800.0 PL=0
MOVL C01256 V=800.0 PL=0
MOVL C01257 V=800.0 PL=0
MOVL C01258 V=800.0 PL=0
MOVL C01259 V=800.0 PL=0
MOVL C01260 V=800.0 PL=0
MOVL C01261 V=800.0 PL=0
MOVL C01262 V=800.0 PL=0
MOVL C01263 V=800.0 PL=0
MOVL C01264 V=800.0 PL=0
MOVL C01265 V=800.0 PL=0
MOVL C01266 V=800.0 PL=0
MOVL C01267 V=800.0 PL=0
MOVL C01268 V=800.0 PL=0
MOVL C01269 V=800.0 PL=0
MOVL C01270 V=800.0 PL=0
MOVL C01271 V=800.0 PL=0
MOVL C01272 V=800.0 PL=0
MOVL C01273 V=800.0 PL=0
MOVL C01274 V=800.0 PL=0
MOVL C01275 V=800.0 PL=0
MOVL C01276 V=800.0 PL=0
MOVL C01277 V=800.0 PL=0
MOVL C01278 V=800.0 PL=0
MOVL C01279 V=800.0 PL=0
MOVL C01280 V=800.0 PL=0
MOVL C01281 V=800.0 PL=0
MOVL C01282 V=800.0 PL=0
MOVL C01283 V=800.0 PL=0
MOVL C01284 V=800.0 PL=0
MOVL C01285 V=800.0 PL=0
MOVL C01286 V=800.0 PL=0
MOVL C01287 V=800.0 PL=0
MOVL C01288 V=800.0 PL=0
MOVL C01289 V=800.0 PL=0
MOVL C01290 V=800.0 PL=0
MOVL C01291 V=800.0 PL=0
MOVL C01292 V=800.0 PL=0
MOVL C01293 V=800.0 PL=0
MOVL C01294 V=800.0 PL=0
MOVL C01295 V=800.0 PL=0
MOVL C01296 V=800.0 PL=0
MOVL C01297 V=800.0 PL=0
MOVL C01298 V=800.0 PL=0
MOVL C01299 V=800.0 PL=0
MOVL C01300 V=800.0 PL=0
MOVL C01301 V=800.0 PL=0
MOVL C01302 V=800.0 PL=0
MOVL C01303 V=800.0 PL=0
MOVL C01304 V=800.0 PL=0
MOVL C01305 V=800.0 PL=0
MOVL C01306 V=800.0 PL=0
MOVL C01307 V=800.0 PL=0
MOVL C01308 V=800.0 PL=0
MOVL C01309 V=800.0 PL=0
MOVL C01310 V=800.0 PL=0
MOVL C01311 V=800.0 PL=0
MOVL C01312 V=800.0 PL=0
MOVL C01313 V=800.0 PL=0
MOVL C01314 V=800.0 PL=0
MOVL C01315 V=800.0 PL=0
MOVL C01316 V=800.0 PL=0
MOVL C01317 V=800.0 PL=0
MOVL C01318 V=800.0 PL=0
MOVL C01319 V=800.0 PL=0
MOVL C01320 V=800.0 PL=0
MOVL C01321 V=800.0 PL=0
MOVL C01322 V=800.0 PL=0
MOVL C01323 V=800.0 PL=0
MOVL C01324 V=800.0 PL=0
MOVL C01325 V=800.0 PL=0
MOVL C01326 V=800.0 PL=0
MOVL C01327 V=800.0 PL=0
MOVL C01328 V=800.0 PL=0
MOVL C01329 V=800.0 PL=0
MOVL C01330 V=800.0 PL=0
MOVL C01331 V=800.0 PL=0
MOVL C01332 V=800.0 PL=0
MOVL C01333 V=800.0 PL=0
MOVL C01334 V=800.0 PL=0
MOVL C01335 V=800.0 PL=0
MOVL C01336 V=800.0 PL=0
MOVL C01337 V=800.0 PL=0
MOVL C01338 V=800.0 PL=0
MOVL C01339 V=800.0 PL=0
MOVL C01340 V=800.0 PL=0
MOVL C01341 V=800.0 PL=0
MOVL C01342 V=800.0 PL=0
MOVL C01343 V=800.0 PL=0
MOVL C01344 V=800.0 PL=0
MOVL C01345 V=800.0 PL=0
MOVL C01346 V=800.0 PL=0
MOVL C01347 V=800.0 PL=0
MOVL C01348 V=800.0 PL=0
MOVL C01349 V=800.0 PL=0
MOVL C01350 V=800.0 PL=0
MOVL C01351 V=800.0 PL=0
MOVL C01352 V=800.0 PL=0
MOVL C01353 V=800.0 PL=0
MOVL C01354 V=800.0 PL=0
MOVL C01355 V=800.0 PL=0
MOVL C01356 V=800.0 PL=0
MOVL C01357 V=800.0 PL=0
MOVL C01358 V=800.0 PL=0
MOVL C01359 V=800.0 PL=0
MOVL C01360 V=800.0 PL=0
MOVL C01361 V=800.0 PL=0
MOVL C01362 V=800.0 PL=0
MOVL C01363 V=800.0 PL=0
MOVL C01364 V=800.0 PL=0
MOVL C01365 V=800.0 PL=0
MOVL C01366 V=800.0 PL=0
MOVL C01367 V=800.0 PL=0
MOVL C01368 V=800.0 PL=0
MOVL C01369 V=800.0 PL=0
MOVL C01370 V=800.0 PL=0
MOVL C01371 V=800.0 PL=0
MOVL C01372 V=800.0 PL=0
MOVL C01373 V=800.0 PL=0
MOVL C01374 V=800.0 PL=0
MOVL C01375 V=800.0 PL=0
MOVL C01376 V=800.0 PL=0
MOVL C01377 V=800.0 PL=0
MOVL C01378 V=800.0 PL=0
MOVL C01379 V=800.0 PL=0
MOVL C01380 V=800.0 PL=0
MOVL C01381 V=800.0 PL=0
MOVL C01382 V=800.0 PL=0
MOVL C01383 V=800.0 PL=0
MOVL C01384 V=800.0 PL=0
MOVL C01385 V=800.0 PL=0
MOVL C01386 V=800.0 PL=0
MOVL C01387 V=800.0 PL=0
MOVL C01388 V=800.0 PL=0
MOVL C01389 V=800.0 PL=0
MOVL C01390 V=800.0 PL=0
MOVL C01391 V=800.0 PL=0
MOVL C01392 V=800.0 PL=0
MOVL C01393 V=800.0 PL=0
MOVL C01394 V=800.0 PL=0
MOVL C01395 V=800.0 PL=0
MOVL C01396 V=800.0 PL=0
MOVL C01397 V=800.0 PL=0
MOVL C01398 V=800.0 PL=0
MOVL C01399 V=800.0 PL=0
MOVL C01400 V=800.0 PL=0
MOVL C01401 V=800.0 PL=0
MOVL C01402 V=800.0 PL=0
MOVL C01403 V=800.0 PL=0
MOVL C01404 V=800.0 PL=0
MOVL C01405 V=800.0 PL=0
MOVL C01406 V=800.0 PL=0
MOVL C01407 V=800.0 PL=0
MOVL C01408 V=800.0 PL=0
MOVL C01409 V=800.0 PL=0
MOVL C01410 V=800.0 PL=0
MOVL C01411 V=800.0 PL=0
MOVL C01412 V=800.0 PL=0
MOVL C01413 V=800.0 PL=0
MOVL C01414 V=800.0 PL=0
MOVL C01415 V=800.0 PL=0
MOVL C01416 V=800.0 PL=0
MOVL C01417 V=800.0 PL=0
MOVL C01418 V=800.0 PL=0
MOVL C01419 V=800.0 PL=0
MOVL C01420 V=800.0 PL=0
MOVL C01421 V=800.0 PL=0
MOVL C01422 V=800.0 PL=0
MOVL C01423 V=800.0 PL=0
MOVL C01424 V=800.0 PL=0
MOVL C01425 V=800.0 PL=0
MOVL C01426 V=800.0 PL=0
MOVL C01427 V=800.0 PL=0
MOVL C01428 V=800.0 PL=0
MOVL C01429 V=800.0 PL=0
MOVL C01430 V=800.0 PL=0
MOVL C01431 V=800.0 PL=0
MOVL C01432 V=800.0 PL=0
MOVL C01433 V=800.0 PL=0
MOVL C01434 V=800.0 PL=0
MOVL C01435 V=800.0 PL=0
MOVL C01436 V=800.0 PL=0
MOVL C01437 V=800.0 PL=0
MOVL C01438 V=800.0 PL=0
MOVL C01439 V=800.0 PL=0
MOVL C01440 V=800.0 PL=0
MOVL C01441 V=800.0 PL=0
MOVL C01442 V=800.0 PL=0
MOVL C01443 V=800.0 PL=0
MOVL C01444 V=800.0 PL=0
MOVL C01445 V=800.0 PL=0
MOVL C01446 V=800.0 PL=0
MOVL C01447 V=800.0 PL=0
MOVL C01448 V=800.0 PL=0
MOVL C01449 V=800.0 PL=0
MOVL C01450 V=800.0 PL=0
MOVL C01451 V=800.0 PL=0
MOVL C01452 V=800.0 PL=0
MOVL C01453 V=800.0 PL=0
MOVL C01454 V=800.0 PL=0
MOVL C01455 V=800.0 PL=0
MOVL C01456 V=800.0 PL=0
MOVL C01457 V=800.0 PL=0
MOVL C01458 V=800.0 PL=0
MOVL C01459 V=800.0 PL=0
MOVL C01460 V=800.0 PL=0
MOVL C01461 V=800.0 PL=0
MOVL C01462 V=800.0 PL=0
MOVL C01463 V=800.0 PL=0
MOVL C01464 V=800.0 PL=0
MOVL C01465 V=800.0 PL=0
MOVL C01466 V=800.0 PL=0
MOVL C01467 V=800.0 PL=0
MOVL C01468 V=800.0 PL=0
MOVL C01469 V=800.0 PL=0
MOVL C01470 V=800.0 PL=0
MOVL C01471 V=800.0 PL=0
MOVL C01472 V=800.0 PL=0
MOVL C01473 V=800.0 PL=0
MOVL C01474 V=800.0 PL=0
MOVL C01475 V=800.0 PL=0
MOVL C01476 V=800.0 PL=0
MOVL C01477 V=800.0 PL=0
MOVL C01478 V=800.0 PL=0
MOVL C01479 V=800.0 PL=0
MOVL C01480 V=800.0 PL=0
MOVL C01481 V=800.0 PL=0
MOVL C01482 V=800.0 PL=0
MOVL C01483 V=800.0 PL=0
MOVL C01484 V=800.0 PL=0
MOVL C01485 V=800.0 PL=0
MOVL C01486 V=800.0 PL=0
MOVL C01487 V=800.0 PL=0
MOVL C01488 V=800.0 PL=0
MOVL C01489 V=800.0 PL=0
MOVL C01490 V=800.0 PL=0
MOVL C01491 V=800.0 PL=0
MOVL C01492 V=800.0 PL=0
MOVL C01493 V=800.0 PL=0
MOVL C01494 V=800.0 PL=0
MOVL C01495 V=800.0 PL=0
MOVL C01496 V=800.0 PL=0
MOVL C01497 V=800.0 PL=0
MOVL C01498 V=800.0 PL=0
MOVL C01499 V=800.0 PL=0
MOVL C01500 V=800.0 PL=0
MOVL C01501 V=800.0 PL=0
MOVL C01502 V=800.0 PL=0
MOVL C01503 V=800.0 PL=0
MOVL C01504 V=800.0 PL=0
MOVL C01505 V=800.0 PL=0
MOVL C01506 V=800.0 PL=0
MOVL C01507 V=800.0 PL=0
MOVL C01508 V=800.0 PL=0
MOVL C01509 V=800.0 PL=0
MOVL C01510 V=800.0 PL=0
MOVL C01511 V=800.0 PL=0
MOVL C01512 V=800.0 PL=0
MOVL C01513 V=800.0 PL=0
MOVL C01514 V=800.0 PL=0
MOVL C01515 V=800.0 PL=0
MOVL C01516 V=800.0 PL=0
MOVL C01517 V=800.0 PL=0
MOVL C01518 V=800.0 PL=0
MOVL C01519 V=800.0 PL=0
MOVL C01520 V=800.0 PL=0
MOVL C01521 V=800.0 PL=0
MOVL C01522 V=800.0 PL=0
MOVL C01523 V=800.0 PL=0
MOVL C01524 V=800.0 PL=0
MOVL C01525 V=800.0 PL=0
MOVL C01526 V=800.0 PL=0
MOVL C01527 V=800.0 PL=0
MOVL C01528 V=800.0 PL=0
MOVL C01529 V=800.0 PL=0
MOVL C01530 V=800.0 PL=0
MOVL C01531 V=800.0 PL=0
MOVL C01532 V=800.0 PL=0
MOVL C01533 V=800.0 PL=0
MOVL C01534 V=800.0 PL=0
MOVL C01535 V=800.0 PL=0
MOVL C01536 V=800.0 PL=0
MOVL C01537 V=800.0 PL=0
MOVL C01538 V=800.0 PL=0
MOVL C01539 V=800.0 PL=0
MOVL C01540 V=800.0 PL=0
MOVL C01541 V=800.0 PL=0
MOVL C01542 V=800.0 PL=0
MOVL C01543 V=800.0 PL=0
MOVL C01544 V=800.0 PL=0
MOVL C01545 V=800.0 PL=0
MOVL C01546 V=800.0 PL=0
MOVL C01547 V=800.0 PL=0
MOVL C01548 V=800.0 PL=0
MOVL C01549 V=800.0 PL=0
MOVL C01550 V=800.0 PL=0
MOVL C01551 V=800.0 PL=0
MOVL C01552 V=800.0 PL=0
MOVL C01553 V=800.0 PL=0
MOVL C01554 V=800.0 PL=0
MOVL C01555 V=800.0 PL=0
MOVL C01556 V=800.0 PL=0
MOVL C01557 V=800.0 PL=0
MOVL C01558 V=800.0 PL=0
MOVL C01559 V=800.0 PL=0
MOVL C01560 V=800.0 PL=0
MOVL C01561 V=800.0 PL=0
MOVL C01562 V=800.0 PL=0
MOVL C01563 V=800.0 PL=0
MOVL C01564 V=800.0 PL=0
MOVL C01565 V=800.0 PL=0
MOVL C01566 V=800.0 PL=0
MOVL C01567 V=800.0 PL=0
MOVL C01568 V=800.0 PL=0
MOVL C01569 V=800.0 PL=0
MOVL C01570 V=800.0 PL=0
MOVL C01571 V=800.0 PL=0
MOVL C01572 V=800.0 PL=0
MOVL C01573 V=800.0 PL=0
MOVL C01574 V=800.0 PL=0
MOVL C01575 V=800.0 PL=0
MOVL C01576 V=800.0 PL=0
MOVL C01577 V=800.0 PL=0
MOVL C01578 V=800.0 PL=0
MOVL C01579 V=800.0 PL=0
MOVL C01580 V=800.0 PL=0
MOVL C01581 V=800.0 PL=0
MOVL C01582 V=800.0 PL=0
MOVL C01583 V=800.0 PL=0
MOVL C01584 V=800.0 PL=0
MOVL C01585 V=800.0 PL=0
MOVL C01586 V=800.0 PL=0
MOVL C01587 V=800.0 PL=0
MOVL C01588 V=800.0 PL=0
MOVL C01589 V=800.0 PL=0
MOVL C01590 V=800.0 PL=0
MOVL C01591 V=800.0 PL=0
MOVL C01592 V=800.0 PL=0
MOVL C01593 V=800.0 PL=0
MOVL C01594 V=800.0 PL=0
MOVL C01595 V=800.0 PL=0
MOVL C01596 V=800.0 PL=0
MOVL C01597 V=800.0 PL=0
MOVL C01598 V=800.0 PL=0
MOVL C01599 V=800.0 PL=0
MOVL C01600 V=800.0 PL=0
MOVL C01601 V=800.0 PL=0
MOVL C01602 V=800.0 PL=0
MOVL C01603 V=800.0 PL=0
MOVL C01604 V=800.0 PL=0
MOVL C01605 V=800.0 PL=0
MOVL C01606 V=800.0 PL=0
MOVL C01607 V=800.0 PL=0
MOVL C01608 V=800.0 PL=0
MOVL C01609 V=800.0 PL=0
MOVL C01610 V=800.0 PL=0
MOVL C01611 V=800.0 PL=0
MOVL C01612 V=800.0 PL=0
MOVL C01613 V=800.0 PL=0
MOVL C01614 V=800.0 PL=0
MOVL C01615 V=800.0 PL=0
MOVL C01616 V=800.0 PL=0
MOVL C01617 V=800.0 PL=0
MOVL C01618 V=800.0 PL=0
MOVL C01619 V=800.0 PL=0
MOVL C01620 V=800.0 PL=0
MOVL C01621 V=800.0 PL=0
MOVL C01622 V=800.0 PL=0
MOVL C01623 V=800.0 PL=0
MOVL C01624 V=800.0 PL=0
MOVL C01625 V=800.0 PL=0
MOVL C01626 V=800.0 PL=0
MOVL C01627 V=800.0 PL=0
MOVL C01628 V=800.0 PL=0
MOVL C01629 V=800.0 PL=0
MOVL C01630 V=800.0 PL=0
MOVL C01631 V=800.0 PL=0
MOVL C01632 V=800.0 PL=0
MOVL C01633 V=800.0 PL=0
MOVL C01634 V=800.0 PL=0
MOVL C01635 V=800.0 PL=0
MOVL C01636 V=800.0 PL=0
MOVL C01637 V=800.0 PL=0
MOVL C01638 V=800.0 PL=0
MOVL C01639 V=800.0 PL=0
MOVL C01640 V=800.0 PL=0
MOVL C01641 V=800.0 PL=0
MOVL C01642 V=800.0 PL=0
MOVL C01643 V=800.0 PL=0
MOVL C01644 V=800.0 PL=0
MOVL C01645 V=800.0 PL=0
MOVL C01646 V=800.0 PL=0
MOVL C01647 V=800.0 PL=0
MOVL C01648 V=800.0 PL=0
MOVL C01649 V=800.0 PL=0
MOVL C01650 V=800.0 PL=0
MOVL C01651 V=800.0 PL=0
MOVL C01652 V=800.0 PL=0
MOVL C01653 V=800.0 PL=0
MOVL C01654 V=800.0 PL=0
MOVL C01655 V=800.0 PL=0
MOVL C01656 V=800.0 PL=0
MOVL C01657 V=800.0 PL=0
MOVL C01658 V=800.0 PL=0
MOVL C01659 V=800.0 PL=0
MOVL C01660 V=800.0 PL=0
MOVL C01661 V=800.0 PL=0
MOVL C01662 V=800.0 PL=0
MOVL C01663 V=800.0 PL=0
MOVL C01664 V=800.0 PL=0
MOVL C01665 V=800.0 PL=0
MOVL C01666 V=800.0 PL=0
MOVL C01667 V=800.0 PL=0
MOVL C01668 V=800.0 PL=0
MOVL C01669 V=800.0 PL=0
MOVL C01670 V=800.0 PL=0
MOVL C01671 V=800.0 PL=0
MOVL C01672 V=800.0 PL=0
MOVL C01673 V=800.0 PL=0
MOVL C01674 V=800.0 PL=0
MOVL C01675 V=800.0 PL=0
MOVL C01676 V=800.0 PL=0
MOVL C01677 V=800.0 PL=0
MOVL C01678 V=800.0 PL=0
MOVL C01679 V=800.0 PL=0
MOVL C01680 V=800.0 PL=0
MOVL C01681 V=800.0 PL=0
MOVL C01682 V=800.0 PL=0
MOVL C01683 V=800.0 PL=0
MOVL C01684 V=800.0 PL=0
MOVL C01685 V=800.0 PL=0
MOVL C01686 V=800.0 PL=0
MOVL C01687 V=800.0 PL=0
MOVL C01688 V=800.0 PL=0
MOVL C01689 V=800.0 PL=0
MOVL C01690 V=800.0 PL=0
MOVL C01691 V=800.0 PL=0
MOVL C01692 V=800.0 PL=0
MOVL C01693 V=800.0 PL=0
MOVL C01694 V=800.0 PL=0
MOVL C01695 V=800.0 PL=0
MOVL C01696 V=800.0 PL=0
MOVL C01697 V=800.0 PL=0
MOVL C01698 V=800.0 PL=0
MOVL C01699 V=800.0 PL=0
MOVL C01700 V=800.0 PL=0
MOVL C01701 V=800.0 PL=0
MOVL C01702 V=800.0 PL=0
MOVL C01703 V=800.0 PL=0
MOVL C01704 V=800.0 PL=0
MOVL C01705 V=800.0 PL=0
MOVL C01706 V=800.0 PL=0
MOVL C01707 V=800.0 PL=0
MOVL C01708 V=800.0 PL=0
MOVL C01709 V=800.0 PL=0
MOVL C01710 V=800.0 PL=0
MOVL C01711 V=800.0 PL=0
MOVL C01712 V=800.0 PL=0
MOVL C01713 V=800.0 PL=0
MOVL C01714 V=800.0 PL=0
MOVL C01715 V=800.0 PL=0
MOVL C01716 V=800.0 PL=0
MOVL C01717 V=800.0 PL=0
MOVL C01718 V=800.0 PL=0
MOVL C01719 V=800.0 PL=0
MOVL C01720 V=800.0 PL=0
MOVL C01721 V=800.0 PL=0
MOVL C01722 V=800.0 PL=0
MOVL C01723 V=800.0 PL=0
MOVL C01724 V=800.0 PL=0
MOVL C01725 V=800.0 PL=0
MOVL C01726 V=800.0 PL=0
MOVL C01727 V=800.0 PL=0
MOVL C01728 V=800.0 PL=0
MOVL C01729 V=800.0 PL=0
MOVL C01730 V=800.0 PL=0
MOVL C01731 V=800.0 PL=0
MOVL C01732 V=800.0 PL=0
MOVL C01733 V=800.0 PL=0
MOVL C01734 V=800.0 PL=0
MOVL C01735 V=800.0 PL=0
MOVL C01736 V=800.0 PL=0
MOVL C01737 V=800.0 PL=0
MOVL C01738 V=800.0 PL=0
MOVL C01739 V=800.0 PL=0
MOVL C01740 V=800.0 PL=0
MOVL C01741 V=800.0 PL=0
MOVL C01742 V=800.0 PL=0
MOVL C01743 V=800.0 PL=0
MOVL C01744 V=800.0 PL=0
MOVL C01745 V=800.0 PL=0
MOVL C01746 V=800.0 PL=0
MOVL C01747 V=800.0 PL=0
MOVL C01748 V=800.0 PL=0
MOVL C01749 V=800.0 PL=0
MOVL C01750 V=800.0 PL=0
MOVL C01751 V=800.0 PL=0
MOVL C01752 V=800.0 PL=0
MOVL C01753 V=800.0 PL=0
MOVL C01754 V=800.0 PL=0
MOVL C01755 V=800.0 PL=0
MOVL C01756 V=800.0 PL=0
MOVL C01757 V=800.0 PL=0
MOVL C01758 V=800.0 PL=0
MOVL C01759 V=800.0 PL=0
MOVL C01760 V=800.0 PL=0
MOVL C01761 V=800.0 PL=0
MOVL C01762 V=800.0 PL=0
MOVL C01763 V=800.0 PL=0
MOVL C01764 V=800.0 PL=0
MOVL C01765 V=800.0 PL=0
MOVL C01766 V=800.0 PL=0
MOVL C01767 V=800.0 PL=0
MOVL C01768 V=800.0 PL=0
MOVL C01769 V=800.0 PL=0
MOVL C01770 V=800.0 PL=0
MOVL C01771 V=800.0 PL=0
MOVL C01772 V=800.0 PL=0
MOVL C01773 V=800.0 PL=0
MOVL C01774 V=800.0 PL=0
MOVL C01775 V=800.0 PL=0
MOVL C01776 V=800.0 PL=0
MOVL C01777 V=800.0 PL=0
MOVL C01778 V=800.0 PL=0
MOVL C01779 V=800.0 PL=0
MOVL C01780 V=800.0 PL=0
MOVL C01781 V=800.0 PL=0
MOVL C01782 V=800.0 PL=0
MOVL C01783 V=800.0 PL=0
MOVL C01784 V=800.0 PL=0
MOVL C01785 V=800.0 PL=0
MOVL C01786 V=800.0 PL=0
MOVL C01787 V=800.0 PL=0
MOVL C01788 V=800.0 PL=0
MOVL C01789 V=800.0 PL=0
MOVL C01790 V=800.0 PL=0
MOVL C01791 V=800.0 PL=0
MOVL C01792 V=800.0 PL=0
MOVL C01793 V=800.0 PL=0
MOVL C01794 V=800.0 PL=0
MOVL C01795 V=800.0 PL=0
MOVL C01796 V=800.0 PL=0
MOVL C01797 V=800.0 PL=0
MOVL C01798 V=800.0 PL=0
MOVL C01799 V=800.0 PL=0
MOVL C01800 V=800.0 PL=0
MOVL C01801 V=800.0 PL=0
MOVL C01802 V=800.0 PL=0
MOVL C01803 V=800.0 PL=0
MOVL C01804 V=800.0 PL=0
MOVL C01805 V=800.0 PL=0
MOVL C01806 V=800.0 PL=0
MOVL C01807 V=800.0 PL=0
MOVL C01808 V=800.0 PL=0
MOVL C01809 V=800.0 PL=0
MOVL C01810 V=800.0 PL=0
MOVL C01811 V=800.0 PL=0
MOVL C01812 V=800.0 PL=0
MOVL C01813 V=800.0 PL=0
MOVL C01814 V=800.0 PL=0
MOVL C01815 V=800.0 PL=0
MOVL C01816 V=800.0 PL=0
MOVL C01817 V=800.0 PL=0
MOVL C01818 V=800.0 PL=0
MOVL C01819 V=800.0 PL=0
MOVL C01820 V=800.0 PL=0
MOVL C01821 V=800.0 PL=0
MOVL C01822 V=800.0 PL=0
MOVL C01823 V=800.0 PL=0
MOVL C01824 V=800.0 PL=0
MOVL C01825 V=800.0 PL=0
MOVL C01826 V=800.0 PL=0
MOVL C01827 V=800.0 PL=0
MOVL C01828 V=800.0 PL=0
MOVL C01829 V=800.0 PL=0
MOVL C01830 V=800.0 PL=0
MOVL C01831 V=800.0 PL=0
MOVL C01832 V=800.0 PL=0
MOVL C01833 V=800.0 PL=0
MOVL C01834 V=800.0 PL=0
MOVL C01835 V=800.0 PL=0
MOVL C01836 V=800.0 PL=0
MOVL C01837 V=800.0 PL=0
MOVL C01838 V=800.0 PL=0
MOVL C01839 V=800.0 PL=0
MOVL C01840 V=800.0 PL=0
MOVL C01841 V=800.0 PL=0
MOVL C01842 V=800.0 PL=0
MOVL C01843 V=800.0 PL=0
MOVL C01844 V=800.0 PL=0
MOVL C01845 V=800.0 PL=0
MOVL C01846 V=800.0 PL=0
MOVL C01847 V=800.0 PL=0
MOVL C01848 V=800.0 PL=0
MOVL C01849 V=800.0 PL=0
MOVL C01850 V=800.0 PL=0
MOVL C01851 V=800.0 PL=0
MOVL C01852 V=800.0 PL=0
MOVL C01853 V=800.0 PL=0
MOVL C01854 V=800.0 PL=0
MOVL C01855 V=800.0 PL=0
MOVL C01856 V=800.0 PL=0
MOVL C01857 V=800.0 PL=0
MOVL C01858 V=800.0 PL=0
MOVL C01859 V=800.0 PL=0
MOVL C01860 V=800.0 PL=0
MOVL C01861 V=800.0 PL=0
MOVL C01862 V=800.0 PL=0
MOVL C01863 V=800.0 PL=0
MOVL C01864 V=800.0 PL=0
MOVL C01865 V=800.0 PL=0
MOVL C01866 V=800.0 PL=0
MOVL C01867 V=800.0 PL=0
MOVL C01868 V=800.0 PL=0
MOVL C01869 V=800.0 PL=0
MOVL C01870 V=800.0 PL=0
MOVL C01871 V=800.0 PL=0
MOVL C01872 V=800.0 PL=0
MOVL C01873 V=800.0 PL=0
MOVL C01874 V=800.0 PL=0
MOVL C01875 V=800.0 PL=0
MOVL C01876 V=800.0 PL=0
MOVL C01877 V=800.0 PL=0
MOVL C01878 V=800.0 PL=0
MOVL C01879 V=800.0 PL=0
MOVL C01880 V=800.0 PL=0
MOVL C01881 V=800.0 PL=0
MOVL C01882 V=800.0 PL=0
MOVL C01883 V=800.0 PL=0
MOVL C01884 V=800.0 PL=0
MOVL C01885 V=800.0 PL=0
MOVL C01886 V=800.0 PL=0
MOVL C01887 V=800.0 PL=0
MOVL C01888 V=800.0 PL=0
MOVL C01889 V=800.0 PL=0
MOVL C01890 V=800.0 PL=0
MOVL C01891 V=800.0 PL=0
MOVL C01892 V=800.0 PL=0
MOVL C01893 V=800.0 PL=0
MOVL C01894 V=800.0 PL=0
MOVL C01895 V=800.0 PL=0
MOVL C01896 V=800.0 PL=0
MOVL C01897 V=800.0 PL=0
MOVL C01898 V=800.0 PL=0
MOVL C01899 V=800.0 PL=0
MOVL C01900 V=800.0 PL=0
MOVL C01901 V=800.0 PL=0
MOVL C01902 V=800.0 PL=0
MOVL C01903 V=800.0 PL=0
MOVL C01904 V=800.0 PL=0
MOVL C01905 V=800.0 PL=0
MOVL C01906 V=800.0 PL=0
MOVL C01907 V=800.0 PL=0
MOVL C01908 V=800.0 PL=0
MOVL C01909 V=800.0 PL=0
MOVL C01910 V=800.0 PL=0
MOVL C01911 V=800.0 PL=0
MOVL C01912 V=800.0 PL=0
MOVL C01913 V=800.0 PL=0
MOVL C01914 V=800.0 PL=0
MOVL C01915 V=800.0 PL=0
MOVL C01916 V=800.0 PL=0
MOVL C01917 V=800.0 PL=0
MOVL C01918 V=800.0 PL=0
MOVL C01919 V=800.0 PL=0
MOVL C01920 V=800.0 PL=0
MOVL C01921 V=800.0 PL=0
MOVL C01922 V=800.0 PL=0
